// TwinCAT 3 PLC project OOP_Curso
// ProgramVersion: 3.1.4023.0
// libraries:
//   Tc2_Standard, * (Beckhoff Automation GmbH)
//   Tc2_System, * (Beckhoff Automation GmbH)
//   Tc2_Utilities, * (Beckhoff Automation GmbH)
//   Tc3_Module, * (Beckhoff Automation GmbH)
// project tree:
//   02_Clases_Y_Objetos/Clase/ Coche.TcPOU
//   02_Clases_Y_Objetos/ _02_Clase_y_Objetos.TcPOU
//   03_Clases_Y_Objetos/Clase/ Coche_3.TcPOU
//   03_Clases_Y_Objetos/ _03_Clase_y_Objetos.TcPOU
//   04_Clases_Y_Objetos/Clase/ fb_tipos_de_datos.TcPOU
//   04_Clases_Y_Objetos/ GVL4.TcGVL, _04_Clases_y_Objetos.TcPOU
//   05_Metodo/ fbreturn5.TcPOU, FB_ejemplo_Method.TcPOU, interface3.TcIO, ST_sample2.TcDUT, _05_Metodo.TcPOU
//   06_Propiedad/ FB_ejemplo_Propiedad.TcPOU, ST_Property.TcDUT, _06_Propiedad.TcPOU
//   07_Herencia_FB/ FB_Hijo.TcPOU (not stored), FB_Padre.TcPOU, Motor.TcPOU (not stored), Pump.TcPOU (not stored), _07_Herencia.TcPOU (not stored)
//   08_Herencia_Estructura_y_Interface/Herencia_Estructura/ ST_1.TcDUT, ST_2.TcDUT, ST_Base1.TcDUT, ST_Sub1.TcDUT, ST_Sub2.TcDUT
//   08_Herencia_Estructura_y_Interface/Herencia_Interface/ FB_Sub1.TcPOU, FB_Sub2.TcPOU, I_Base1.TcIO, I_Base2.TcIO, I_Sub1.TcIO, I_Sub2.TcIO
//   08_Herencia_Estructura_y_Interface/ _08_Herencia_Estructura_y_Interface.TcPOU
//   09_THIS_SUPER/SUPER/ FB_1.TcPOU, FB_Base.TcPOU
//   09_THIS_SUPER/THIS/ FB_A.TcPOU, FB_B.TcPOU, F_FunA.TcPOU
//   09_THIS_SUPER/ _09_THIS_SUPER.TcPOU
//   10_Interface/Interface1/ FB_Sensor.TcPOU, I_Sensor.TcIO
//   10_Interface/Interface2/ FB_TestA.TcPOU, FB_TestB.TcPOU, ITF_MyTest.TcIO, myFC.TcPOU
//   10_Interface/ _10_Interface.TcPOU
//   11_Puntero_y_Referencia/ Fc_AreaCalcPoint.TcPOU, Fc_AreaCalcRef.TcPOU, Fc_AreaCalcVal.TcPOU, Fc_AverageReferencia.TcPOU, Fc_AverageValues.TcPOU, SR_Main_01.TcPOU, SR_Main_02.TcPOU, SR_Main_03.TcPOU, SR_Main_04.TcPOU, stMotorCtrl.TcDUT, st_Rectangulo.TcDUT, _11_Puntero_y_Referencia.TcPOU
//   13_FB_Abstracto_vs_Interface/1_FB_Abstracto/ ClassDiagram.TcCD (not stored), FB_ContractEmployee.TcPOU (not stored), FB_Employee.TcPOU (not stored), FB_FullTimeEmployee.TcPOU, _13_1_Main_Abstract.TcPOU
//   13_FB_Abstracto_vs_Interface/2_Interfaz/ ClassDiagram_1.TcCD (not stored), FB_ContractEmployee_1.TcPOU (not stored), FB_FullTimeEmployee_1.TcPOU (not stored), I_Employee.TcIO (not stored), _13_2_Main_Interfaz.TcPOU
//   13_FB_Abstracto_vs_Interface/3_Combinacion/ ClassDiagram_2.TcCD (not stored), FB_ContractEmployee_2.TcPOU, FB_Employee_1.TcPOU (not stored), FB_FullTimeEmployee_2.TcPOU (not stored), I_Employee_1.TcIO (not stored), _13_3_Main_Combinacion.TcPOU
//   12_Concepto Keyword Abstract/ AbstractLoadCell.TcPOU, AbstractLogger.TcPOU, ConcreteADSLogger.TcPOU, ConcreteCSVLogger.TcPOU, ConcreteLoadCell.TcPOU, _12_Concepto_Keyword_Abstract.TcPOU
//   14_Interface_Fluida/14_1/ FB_Calculate.TcPOU, I_Calculate.TcIO
//   14_Interface_Fluida/14_2/ FB_Calcul.TcPOU, I_Clear.TcIO, I_Operation.TcIO, I_SetNumber.TcIO
//   14_Interface_Fluida/ _14_Interface_Fluida.TcPOU
//   15_Interface_vs_Herencia/ ClassDiagram_3.TcCD (not stored), FB_NivelSensor.TcPOU, FB_Pump.TcPOU, I_Analog.TcIO, I_Run.TcIO, FB_UltraSonicSensor.TcPOU, FB_VFD.TcPOU, _15_Interface_vs_Herencia.TcPOU
//   16_17_Interface_vs_Herencia/ FB_MyLight1.TcPOU, _16_Interface_vs_Herencia.TcPOU (not stored)
//   16_17_Interface_vs_Herencia/PLC-Library/Clases/ FB_DelayedLight.TcPOU (not stored), FB_DimmingLight.TcPOU (not stored), FB_Light.TcPOU, FB_RoomController.TcPOU (not stored)
//   16_17_Interface_vs_Herencia/PLC-Library/ ClassDiagram_4.TcCD (not stored), FB_MyLight.TcPOU
//   16_17_Interface_vs_Herencia/PLC-Library/Interfaces/ I_Delayable.TcIO, I_Dimmable.TcIO (not stored), I_Light.TcIO (not stored)
//   16_17_Interface_vs_Herencia/Tests/ P_DelayedLight_Test_CFC.TcPOU (not stored), P_DelayedLight_Test_ST.TcPOU (not stored), P_DimmingLight_Test_CFC.TcPOU, P_DimmingLight_Test_ST.TcPOU (not stored), P_Light_Test_CFC.TcPOU, P_Light_Test_ST.TcPOU, P_MyLight_Test_CFC.TcPOU, P_MyLight_Test_ST.TcPOU, P_RoomController_Test_CFC.TcPOU, P_RoomController_Test_ST.TcPOU
//   17_Otros_Operadores_1/ ST_Estructura.TcDUT (not stored), _17_Otros_Operadores1.TcPOU
//   18_Otros_Operadores_2/TestAndSet/ GVL.TcGVL, TestAndSet1.TcPOU
//   18_Otros_Operadores_2/ _18_Otros_Operadores2.TcPOU
//   18_Otros_Operadores_2/__QUERYPOINTER/ FB_Variante.TcPOU, I_Base.TcIO, I_Derived.TcIO, QUERYPOINTER.TcPOU
//   18_Otros_Operadores_2/__TRY__CATCH/ GVL_Exc.TcGVL, F_SaveExceptionCode.TcPOU, TRY_CATCH.TcPOU
//   18_Otros_Operadores_2/__VARINFO/ VARINFO.TcPOU
//   19_ExST/ _19_ExST.TcPOU
//   24_SOLID_SRP/Clases_SRP/ FB_Empleado.TcPOU (not stored), FB_RegistroDeTiempo.TcPOU
//   24_SOLID_SRP/ Class Diagram_SOLID_SRP.TcCD (not stored), _24_SOLID_SRP.TcPOU
//   24_SOLID_SRP/Estructuras_SRP/ ST_Empleado.TcDUT (not stored), ST_Horario.TcDUT, ST_RegistroDeTiempoEmpleado.TcDUT
//   25_SOLID_OCP/Clases_OCP/ FB_Coche.TcPOU, FB_Moto.TcPOU, FB_Vehiculo.TcPOU
//   25_SOLID_OCP/ Class Diagram_SOLID_OCP.TcCD (not stored), _25_SOLID_OCP.TcPOU
//   26_SOLID_LSP/Clases_LSP/ Coche1.TcPOU, Conductor.TcPOU, Moto1.TcPOU, Vehiculo.TcPOU
//   26_SOLID_LSP/ Class Diagram_SOLID_LSP.TcCD (not stored), _26_SOLID_LSP.TcPOU
//   26_SOLID_LSP/Interfaces_LSP/ I_Mover.TcIO
//   27_SOLID_ISP/Clases_ISP/ Aguila.TcPOU, Avestruz.TcPOU, Pato.TcPOU
//   27_SOLID_ISP/ Class Diagram_SOLID_ISP.TcCD (not stored), _27_SOLID_ISP.TcPOU
//   27_SOLID_ISP/Interfaces_ISP/ I_AveCorredora.TcIO, I_AveNadadora.TcIO, I_AveVoladora.TcIO
//   28_SOLID_DIP/Clases_DIP/ ConexionEthernet.TcPOU, ConexionSerial.TcPOU, Dispositivo.TcPOU
//   28_SOLID_DIP/ ClassDiagram_SOLID_DIP.TcCD (not stored), _28_SOLID_DIP.TcPOU
//   28_SOLID_DIP/Interfaces_DIP/ I_Conexion.TcIO
//   30_UML_ClassDiagram/ 30_UML_ClassDiagram.TcCD (not stored), GVL_1.TcGVL, ITF_Profesor.TcIO, Persona.TcPOU, Profesor.TcPOU
//   31_UML_relaciones/ ClassDiagram_UML_Relaciones.TcCD (not stored), Corazon.TcPOU, Hombre.TcPOU, Humano.TcPOU, I_Humano.TcIO, Sangre.TcPOU
//   32_UML_StateChart/32_VISU/ _32_Visualization.TcVIS
//   32_UML_StateChart/ Kaffemaschine.TcPOU
//   32_UML_StateChart/32_POUs/ FB_UML_SC.TcPOU, _32_MAIN.TcPOU
//   / Gestor de visualización.TcVMO (not stored), GlobalTextList.TcGTLO, PlcTask.TcTTO
//   _MAIN/ MAIN.TcPOU
// real-time tasks:
//   TASK PlcTask: cycle T#10ms, priority 20, ADS port 350

CONFIGURATION OOP_Curso
    RESOURCE PLC ON TwinCAT3
        TASK PlcTask(INTERVAL := T#10ms, PRIORITY := 20);
        PROGRAM MAIN WITH PlcTask : MAIN;
    END_RESOURCE
END_CONFIGURATION

// ---- 05_Metodo/ST_sample2.TcDUT
TYPE ST_sample2 :
STRUCT
	bbool	: BOOL;
	bVar 	: BOOL;
    nVar 	: INT;
	rreal 	: REAL;
	sstring : STRING;
END_STRUCT
END_TYPE

// ---- 06_Propiedad/ST_Property.TcDUT
TYPE ST_Property :
STRUCT
	b1,b2,b3 : BOOL;
	r1,r2,r3 : REAL;	
END_STRUCT
END_TYPE

// ---- 08_Herencia_Estructura_y_Interface/Herencia_Estructura/ST_1.TcDUT
TYPE ST_1:
STRUCT
	sStruct : ST_2;
	sstring : STRING(80);
END_STRUCT
END_TYPE

// ---- 08_Herencia_Estructura_y_Interface/Herencia_Estructura/ST_2.TcDUT
TYPE ST_2 :
STRUCT
	bBool : BOOL;
END_STRUCT
END_TYPE

// ---- 08_Herencia_Estructura_y_Interface/Herencia_Estructura/ST_Base1.TcDUT
TYPE ST_Base1 :
STRUCT
	bBool1: BOOL;
	iINT : INT;
	rReal : REAL;	
END_STRUCT
END_TYPE

// ---- 08_Herencia_Estructura_y_Interface/Herencia_Estructura/ST_Sub1.TcDUT
TYPE ST_Sub1 EXTENDS ST_Base1:
STRUCT
	ttime :TIME;
	tton  : TON;
END_STRUCT
END_TYPE

// ---- 08_Herencia_Estructura_y_Interface/Herencia_Estructura/ST_Sub2.TcDUT
TYPE ST_Sub2 EXTENDS ST_Sub1 :
STRUCT
	bBool2: BOOL;
END_STRUCT
END_TYPE

// ---- 11_Puntero_y_Referencia/stMotorCtrl.TcDUT
TYPE stMotorCtrl :
STRUCT
	rTpoAcelDecel :REAL; // Tiempo para acelerar/decelerar hasta alcanazar la velocidad.
	rVelRpm       :REAL; // Velocidad en RPM.
	xMotorOff     :BOOL; // Bit de paro ON.
	xMotorOn      :BOOL   ; // Bit de marcha OFF.	
END_STRUCT
END_TYPE

// ---- 11_Puntero_y_Referencia/st_Rectangulo.TcDUT
TYPE st_Rectangulo :
STRUCT
   rASide    	: REAL; // Parámetro de entrada que contiene el lado A del rectangulo.
   rBSide    	: REAL; // Parámetro de entrada que contiene el lado B del rectangulo.	
   rArea		: REAL; // Valor del area
END_STRUCT
END_TYPE

// ---- 24_SOLID_SRP/Estructuras_SRP/ST_Horario.TcDUT
TYPE ST_Horario :
STRUCT
	HoraEntrada : DATE_AND_TIME;
    HoraSalida : DATE_AND_TIME;
END_STRUCT
END_TYPE

// ---- 24_SOLID_SRP/Estructuras_SRP/ST_RegistroDeTiempoEmpleado.TcDUT
TYPE ST_RegistroDeTiempoEmpleado :
STRUCT
	stEmpleado : ST_Empleado; // Datos de la función Empleado
    stHorario  : ST_Horario;
END_STRUCT
END_TYPE

// ---- 04_Clases_Y_Objetos/GVL4.TcGVL
//{attribute 'qualified_only'}
VAR_GLOBAL
	 nVarExt1 : INT; // 1st external variable
END_VAR

// ---- 18_Otros_Operadores_2/TestAndSet/GVL.TcGVL
{attribute 'qualified_only'}
VAR_GLOBAL
    bGlobalTestFlag : BOOL;
END_VAR

// ---- 18_Otros_Operadores_2/__TRY__CATCH/GVL_Exc.TcGVL
{attribute 'qualified_only'}
VAR_GLOBAL CONSTANT
    cMaxExc            : UINT := 10;
END_VAR
VAR_GLOBAL
    nExcIndex          : UINT;
    aExceptionHistory  : ARRAY[0..cMaxExc] OF __SYSTEM.ExceptionCode;
END_VAR

// ---- 30_UML_ClassDiagram/GVL_1.TcGVL
{attribute 'qualified_only'}
VAR_GLOBAL
	variable1 : BOOL;
	VarInt: INT;
END_VAR

// ---- 05_Metodo/interface3.TcIO
INTERFACE interface3

METHOD itf_metodo : BOOL
VAR_INPUT
END_VAR
END_METHOD

PROPERTY itf_propiedad : real
GET
END_GET
SET
END_SET
END_PROPERTY

END_INTERFACE

// ---- 08_Herencia_Estructura_y_Interface/Herencia_Interface/I_Base1.TcIO
INTERFACE I_Base1

METHOD metodo_base1 : BOOL
VAR_INPUT
END_VAR
END_METHOD

PROPERTY Prop_base1 : bool
GET
END_GET
SET
END_SET
END_PROPERTY

END_INTERFACE

// ---- 08_Herencia_Estructura_y_Interface/Herencia_Interface/I_Base2.TcIO
INTERFACE I_Base2

METHOD metodo_base2 : BOOL
VAR_INPUT
END_VAR
END_METHOD

PROPERTY Prop_base2 : bool
GET
END_GET
SET
END_SET
END_PROPERTY

END_INTERFACE

// ---- 08_Herencia_Estructura_y_Interface/Herencia_Interface/I_Sub1.TcIO
INTERFACE I_Sub1 EXTENDS I_Base1, I_Base2

METHOD metodo_sub1 : BOOL
VAR_INPUT
END_VAR
END_METHOD

PROPERTY Prop_sub1 : BOOL
GET
END_GET
SET
END_SET
END_PROPERTY

END_INTERFACE

// ---- 08_Herencia_Estructura_y_Interface/Herencia_Interface/I_Sub2.TcIO
INTERFACE I_Sub2 EXTENDS I_Sub1

METHOD metodo_sub2 : BOOL
VAR_INPUT
END_VAR
END_METHOD

PROPERTY Prop_sub2 : BOOL
GET
END_GET
SET
END_SET
END_PROPERTY

END_INTERFACE

// ---- 10_Interface/Interface1/I_Sensor.TcIO
INTERFACE I_Sensor

PROPERTY Calibrado : BOOL
GET
END_GET
END_PROPERTY

METHOD Calibrar
END_METHOD

PROPERTY Consigna : REAL
SET
END_SET
END_PROPERTY


METHOD Descalibrar
END_METHOD

METHOD LeerValor : INT
END_METHOD

PROPERTY Temperatura : REAL
GET
END_GET
END_PROPERTY

END_INTERFACE

// ---- 10_Interface/Interface2/ITF_MyTest.TcIO
INTERFACE ITF_MyTest

METHOD METH1 : BOOL
VAR_INPUT
END_VAR
END_METHOD

METHOD METH2 : STRING
VAR_INPUT
END_VAR
END_METHOD

METHOD METH3 : REAL
VAR_INPUT
END_VAR
END_METHOD

PROPERTY Prop1 : BOOL
GET
END_GET
SET
END_SET
END_PROPERTY

PROPERTY Prop2 : REAL
GET
END_GET
SET
END_SET
END_PROPERTY

PROPERTY Prop3 : STRING
GET
END_GET
SET
END_SET
END_PROPERTY

END_INTERFACE

// ---- 14_Interface_Fluida/14_1/I_Calculate.TcIO
INTERFACE I_Calculate

METHOD Clear : I_Calculate
END_METHOD

METHOD DecreaseBy : I_Calculate
VAR_INPUT
	lDecreaseBy : REAL;
END_VAR
END_METHOD

METHOD DivideBy : I_Calculate
VAR_INPUT
	lDivideBy : REAL;
END_VAR
END_METHOD

METHOD GetResult : LREAL
VAR_INPUT
END_VAR
END_METHOD

METHOD IncreaseBy : I_Calculate
VAR_INPUT
	lIncreaseBy : REAL;
END_VAR
END_METHOD

METHOD MultiplyBy : I_Calculate
VAR_INPUT
	lMultiplyBy : REAL;
END_VAR
END_METHOD

METHOD SetNumber : I_Calculate
VAR_INPUT
	lNumber : LREAL;
END_VAR
END_METHOD

END_INTERFACE

// ---- 14_Interface_Fluida/14_2/I_Clear.TcIO
INTERFACE I_Clear

METHOD Clear : I_SetNumber
END_METHOD

END_INTERFACE

// ---- 14_Interface_Fluida/14_2/I_Operation.TcIO
INTERFACE I_Operation EXTENDS I_SetNumber


METHOD DecreaseBy : I_Operation
VAR_INPUT
	lDecreaseBy : REAL;
END_VAR
END_METHOD


METHOD DivideBy : I_Operation
VAR_INPUT
	lDivideBy : REAL;
END_VAR
END_METHOD


METHOD GetResult : LREAL
END_METHOD

METHOD IncreaseBy : I_Operation
VAR_INPUT
	lIncreaseBy : REAL;
END_VAR
END_METHOD


METHOD MultiplyBy : I_Operation
VAR_INPUT
	lMultiplyBy : REAL;
END_VAR
END_METHOD

END_INTERFACE

// ---- 14_Interface_Fluida/14_2/I_SetNumber.TcIO
INTERFACE I_SetNumber

METHOD SetNumber : I_Operation
VAR_INPUT
	lNumber : LREAL;
END_VAR
END_METHOD

END_INTERFACE

// ---- 15_Interface_vs_Herencia/I_Analog.TcIO
INTERFACE I_Analog

PROPERTY AnalogSignal : INT
GET
END_GET
SET
END_SET
END_PROPERTY

METHOD Scale : BOOL
VAR_INPUT
END_VAR
END_METHOD

PROPERTY ScaledAnalog : INT
GET
END_GET
SET
END_SET
END_PROPERTY

END_INTERFACE

// ---- 15_Interface_vs_Herencia/I_Run.TcIO
INTERFACE I_Run

PROPERTY Coil : BOOL
GET
END_GET
SET
END_SET
END_PROPERTY

METHOD Start : BOOL
VAR_INPUT
END_VAR
END_METHOD

METHOD Stop : BOOL
VAR_INPUT
END_VAR
END_METHOD

END_INTERFACE

// ---- 16_17_Interface_vs_Herencia/PLC-Library/Interfaces/I_Delayable.TcIO
INTERFACE I_Delayable EXTENDS __SYSTEM.IQueryInterface

PROPERTY tOffDelay : TIME
GET
END_GET
SET
END_SET
END_PROPERTY

PROPERTY tOnDelay : TIME
GET
END_GET
SET
END_SET
END_PROPERTY

END_INTERFACE

// ---- 18_Otros_Operadores_2/__QUERYPOINTER/I_Base.TcIO
INTERFACE I_Base EXTENDS __SYSTEM.IQueryInterface

METHOD Base : BOOL
VAR_INPUT
END_VAR
END_METHOD

END_INTERFACE

// ---- 18_Otros_Operadores_2/__QUERYPOINTER/I_Derived.TcIO
INTERFACE I_Derived EXTENDS I_Base

METHOD Derived : BOOL
VAR_INPUT
END_VAR
END_METHOD

END_INTERFACE

// ---- 26_SOLID_LSP/Interfaces_LSP/I_Mover.TcIO
INTERFACE I_Mover

METHOD Mover : REAL
VAR_INPUT
	Velocidad_Deseada : REAL;
END_VAR
END_METHOD

END_INTERFACE

// ---- 27_SOLID_ISP/Interfaces_ISP/I_AveCorredora.TcIO
INTERFACE I_AveCorredora

METHOD Correr : BOOL
END_METHOD

END_INTERFACE

// ---- 27_SOLID_ISP/Interfaces_ISP/I_AveNadadora.TcIO
INTERFACE I_AveNadadora

METHOD Nadar : BOOL
END_METHOD

END_INTERFACE

// ---- 27_SOLID_ISP/Interfaces_ISP/I_AveVoladora.TcIO
INTERFACE I_AveVoladora

METHOD Volar : BOOL
END_METHOD

END_INTERFACE

// ---- 28_SOLID_DIP/Interfaces_DIP/I_Conexion.TcIO
INTERFACE I_Conexion

METHOD EstablecerConexion : BOOL
VAR_INPUT
END_VAR
END_METHOD

END_INTERFACE

// ---- 30_UML_ClassDiagram/ITF_Profesor.TcIO
INTERFACE ITF_Profesor

METHOD Fichar
VAR_INPUT
END_VAR
END_METHOD

PROPERTY Salida : int
GET
END_GET
SET
END_SET
END_PROPERTY

END_INTERFACE

// ---- 31_UML_relaciones/I_Humano.TcIO
INTERFACE I_Humano

METHOD Correr
VAR_INPUT
END_VAR
END_METHOD

PROPERTY Nombre : STRING
GET
END_GET
SET
END_SET
END_PROPERTY

END_INTERFACE

// ---- _MAIN/MAIN.TcPOU
PROGRAM MAIN
VAR
END_VAR

// Video de Youtube 02:
_02_Clase_y_Objetos();

// Video de Youtube 03:
_03_Clase_y_Objetos();

// Video de Youtube 04:
_04_Clases_y_Objetos();

// Video de Youtube 05;
_05_Metodo();

// Video de Youtube 06;
_06_Propiedad();

// Video de Youtube 07;
_07_Herencia();

// Video de Youtube 08;
_08_Herencia_Estructura_y_Interface();

// Video de Youtube 09;
_09_THIS_SUPER();

// Video de Youtube 10;
_10_Interface();

// Video de Youtube 11;
_11_Puntero_y_Referencia();

// Video de Youtube 12;
_12_Concepto_Keyword_Abstract();

// Video de Youtube 13;
_13_1_Main_Abstract();
_13_2_Main_Interfaz();
_13_3_Main_Combinacion();

// Video de Youtube 14;
_14_Interface_Fluida();

// Video de Youtube 15:
_15_Interface_vs_Herencia();

// Video de Youtube 16:
_16_Interface_vs_Herencia();

// Video de Youtube 17:
_17_Otros_Operadores1();

// Video de Youtube 18:
_18_Otros_Operadores2();

// Video de Youtube 19:
_19_ExST();

// Video de Youtube 24
_24_SOLID_SRP();

// Video de Youtube 25
_25_SOLID_OCP();

// Video de Youtube 26
_26_SOLID_LSP();

// Video de Youtube 27
_27_SOLID_ISP();

// Video de Youtube 28
_28_SOLID_DIP();

// Video de Youtube 32
_32_MAIN();

END_PROGRAM

// ---- 02_Clases_Y_Objetos/_02_Clase_y_Objetos.TcPOU
PROGRAM _02_Clase_y_Objetos
VAR
	// tenemos la Clase Coche y la instanciamos y obtenemos los Objetos: Mercedes, Bmw y Audi.
	Mercedes : Coche;
	Bmw : Coche;
	Audi: Coche;
	
	Color : STRING;
	Marca : STRING;
	
	Acelerar : BOOL;
	Conducir:  BOOL;
	Frenar  : BOOL;
	
	
END_VAR

//Objeto Mercedes
//llamadas a sus métodos.
IF Acelerar THEN
	Mercedes.Acelerar();
	Acelerar := FALSE;
END_IF

IF Conducir THEN
	Mercedes.Conducir();
	Conducir := FALSE;
END_IF

IF Frenar THEN
	Mercedes.Frenar();
	Frenar := FALSE;
END_IF

//llamadas a sus propiedades.
Mercedes.Marca := 'Mercedes';
Mercedes.Color := 'Negro';
Color := Mercedes.Color;

END_PROGRAM

// ---- 02_Clases_Y_Objetos/Clase/Coche.TcPOU
FUNCTION_BLOCK Coche
VAR_INPUT 
END_VAR
VAR_OUTPUT
END_VAR
VAR
	_Marca : STRING;
	_Color : STRING;
	accion : STRING;
END_VAR

METHOD PUBLIC Acelerar
accion := 'acelerar';
END_METHOD

PROPERTY PUBLIC Color : STRING
GET
Color := _Color;
END_GET
SET
_Color := Color;
END_SET
END_PROPERTY

METHOD PUBLIC Conducir
accion := 'conducir';
END_METHOD

METHOD PUBLIC Frenar
accion := 'frenar';
END_METHOD

PROPERTY PUBLIC Marca : STRING
GET
Marca := _Marca;
END_GET
SET
_Marca := Marca;
END_SET
END_PROPERTY

END_FUNCTION_BLOCK

// ---- 03_Clases_Y_Objetos/_03_Clase_y_Objetos.TcPOU
PROGRAM _03_Clase_y_Objetos
VAR
	// tenemos la Clase Coche y la instanciamos y obtenemos los Objetos: Mercedes, Bmw y Audi.
	Mercedes : Coche_3(Marca:= 'Mercedes', Color := 'Azul');
	
	Color : STRING;
	Marca : STRING;
	
	Acelerar : BOOL;
	Conducir:  BOOL;
	Frenar  : BOOL;
	
	CambiarColor : BOOL;
END_VAR

//Objeto Mercedes
//llamadas a sus métodos.
IF Acelerar THEN
	Mercedes.Acelerar();
	Acelerar := FALSE;
END_IF

IF Conducir THEN
	Mercedes.Conducir();
	Conducir := FALSE;
END_IF

IF Frenar THEN
	Mercedes.Frenar();
	Frenar := FALSE;
END_IF

//llamadas a sus propiedades.
//Mercedes.Marca := 'Mercedes';
IF CambiarColor THEN
	Mercedes.Color := 'Negro';
	CambiarColor := FALSE;
END_IF

Color := Mercedes.Color;

END_PROGRAM

// ---- 03_Clases_Y_Objetos/Clase/Coche_3.TcPOU
FUNCTION_BLOCK Coche_3
VAR_INPUT
	bInput : BOOL;
END_VAR
VAR_OUTPUT
	bOutput : BOOL;
END_VAR
VAR_IN_OUT
	bInOut : BOOL;
END_VAR
VAR
	_Marca : STRING;
	_Color : STRING;
	accion : STRING;
END_VAR

METHOD PUBLIC Acelerar
accion := 'acelerar';
END_METHOD

PROPERTY PUBLIC Color : STRING
GET
Color := _Color;
END_GET
SET
_Color := Color;
END_SET
END_PROPERTY

METHOD PUBLIC Conducir
accion := 'conducir';
END_METHOD

METHOD FB_exit : BOOL
VAR_INPUT
	bInCopyCode : BOOL; // if TRUE, the exit method is called for exiting an instance that is copied afterwards (online change).
END_VAR
END_METHOD

METHOD FB_init : BOOL
VAR_INPUT
	bInitRetains : BOOL; // if TRUE, the retain variables are initialized (warm start / cold start)
	bInCopyCode : BOOL;  // if TRUE, the instance afterwards gets moved into the copy code (online change)
	Marca        : STRING;
	Color        : STRING;
END_VAR
THIS^._Marca := Marca;
THIS^._Color := Color;
END_METHOD

METHOD FB_reinit : BOOL
VAR_INPUT
END_VAR
END_METHOD

METHOD PUBLIC Frenar
accion := 'frenar';
END_METHOD

PROPERTY PUBLIC Marca : STRING
GET
Marca := _Marca;
END_GET
SET
_Marca := Marca;
END_SET
END_PROPERTY

END_FUNCTION_BLOCK

// ---- 04_Clases_Y_Objetos/_04_Clases_y_Objetos.TcPOU
PROGRAM _04_Clases_y_Objetos
VAR
	fb :fb_tipos_de_datos;
	binput : BOOL;
	in_out1 : LINT;
	in_out_constant1 : DINT := 10;
END_VAR


fb(
//	binput:= binput, 
//	binput2:= , 
//	output1=> , 
	in_out1:= in_out1, 
	in_out_constant1:= in_out_constant1 );

END_PROGRAM

// ---- 04_Clases_Y_Objetos/Clase/fb_tipos_de_datos.TcPOU
FUNCTION_BLOCK fb_tipos_de_datos
VAR_INPUT
	binput : BOOL;
END_VAR
VAR_INPUT
	binput2 : BOOL;
END_VAR
VAR_OUTPUT
	output1 : REAL;
END_VAR
VAR_IN_OUT
	in_out1 : LINT;
END_VAR
VAR_IN_OUT CONSTANT
	in_out_constant1 : DINT;
END_VAR
VAR
	var1 : STRING;
END_VAR
VAR_TEMP
	temp1 : ULINT;
END_VAR
VAR_STAT
    nVarStat1 : INT;
	aarray  : ARRAY[1..n] OF INT;
END_VAR
VAR_EXTERNAL
    nVarExt1 : INT; // 1st external variable
END_VAR
VAR PERSISTENT
    nVarPers1 : DINT; (* 1. Persistent variable *)
    bVarPers2 : BOOL; (* 2. Persistent variable *)
END_VAR
VAR RETAIN
    nRem1 : INT;
END_VAR
VAR CONSTANT
	n : INT:= 10;
END_VAR

END_FUNCTION_BLOCK

// ---- 05_Metodo/_05_Metodo.TcPOU
PROGRAM _05_Metodo
VAR
	fbejemplo_metodo : FB_ejemplo_Method;
	
	bPonerAUnobBoolfb : BOOL;
	bPonerACerobBoolfb: BOOL;
	
	bBool : BOOL;
	statusbBool : BOOL;
	bPonerAUnobBool : BOOL;
	bPonerACerobBool: BOOL;
	
	nSingleGet  : INT;
    stGet       : ST_Sample2;    
    bSet        : BOOL;
    stSet       : ST_Sample2;
	
	counter : INT;
	outvarcounter: INT;
END_VAR

IF 	bPonerAUnobBoolfb THEN
	bPonerAUnobBoolfb := FALSE;
	fbejemplo_metodo.metodo1_a_Uno_bBool();	
END_IF


IF 	bPonerACerobBoolfb THEN
	bPonerACerobBoolfb := FALSE;
	fbejemplo_metodo.metodo1_a_cero_bBool();
END_IF


IF 	bPonerAUnobBool THEN
	bPonerAUnobBool := FALSE;
	statusbBool := fbejemplo_metodo.metodo1_a_Uno_InOut(bBool);
END_IF

IF 	bPonerACerobBool THEN
	bPonerACerobBool := FALSE;
	statusbBool := fbejemplo_metodo.metodo1_a_Cero_InOut(bBool);
END_IF

// ejemplo para declarar variables lo mas cerca posible del metodo: declaración dentro del metodo de variable con VAR_INST :
counter := fbejemplo_metodo.Metodo4_VarInst(outvarcounter=>outvarcounter);

// Set and Get
IF bSet THEN  
	nSingleGet := fbejemplo_metodo.metodo2_struct(stSet).nVar;
	stGet      := fbejemplo_metodo.metodo2_struct(stSet);
	bSet            := FALSE;
END_IF

END_PROGRAM

// ---- 05_Metodo/FB_ejemplo_Method.TcPOU
FUNCTION_BLOCK FB_ejemplo_Method
VAR_INPUT
END_VAR
VAR_OUTPUT
END_VAR
VAR
	bBool : BOOL;
	ststruct : ST_sample2;
	fb5 : fbreturn5;
END_VAR

METHOD metodo0_Declaracion_variables
VAR_INPUT
	binput : BOOL;
END_VAR
VAR_INPUT
	binput2 : BOOL;
END_VAR
VAR_OUTPUT
	output1 : REAL;
END_VAR
VAR_IN_OUT
	in_out1 : LINT;
END_VAR
VAR_IN_OUT CONSTANT
	in_out_constant1 : DINT;
END_VAR
VAR
	var1 : STRING;
END_VAR
//!!! no se pueden declarar variables TEMPORALES dentro de la zona de declaración de variables del método!!!
//VAR_TEMP
//	temp1 : ULINT;
//END_VAR
VAR_INST
	counter : INT;
END_VAR
VAR_STAT
    nVarStat1 : INT;
	aarray  : ARRAY[1..n] OF INT;
END_VAR
VAR_EXTERNAL
    nVarExt1 : INT; // 1st external variable
END_VAR
//!!! no se pueden declarar variables PERSISTENT ni RETAIN dentro de la zona de declaración de variables del método!!!
//VAR PERSISTENT
//    nVarPers1 : DINT; (* 1. Persistent variable *)
//    bVarPers2 : BOOL; (* 2. Persistent variable *)
//END_VAR
//VAR RETAIN
//    nRem1 : INT;
//END_VAR
VAR CONSTANT
	n : INT:= 10;
END_VAR
END_METHOD

METHOD metodo1_a_Cero_bBool
THIS^.bBool := false;
END_METHOD

METHOD metodo1_a_Cero_InOut : bool
VAR_IN_OUT
	bBool : BOOL;
END_VAR
// Método que pone a 0 la variable definida en in_Out
bBool := FALSE;
// return value bBOOL
metodo1_a_Cero_InOut := FALSE;
END_METHOD

METHOD metodo1_a_Uno_bBool
THIS^.bBool := true;
END_METHOD

METHOD metodo1_a_Uno_InOut : BOOL
VAR_IN_OUT
	bBool : BOOL;
END_VAR
// Método que pone a 1 la variable definida en in_Out
bBool := TRUE;
// return value bBOOL
metodo1_a_Uno_InOut := TRUE;
END_METHOD

METHOD PUBLIC metodo2_struct : REFERENCE TO ST_sample2
VAR_INPUT
	st_struct : ST_sample2;
END_VAR


THIS^.ststruct := st_struct;

metodo2_struct REF= THIS^.ststruct;
END_METHOD

METHOD PRIVATE metodo3_interface : interface3
VAR_INPUT
END_VAR
END_METHOD

METHOD Metodo4_VarInst : INT
VAR_OUTPUT
	outvarcounter : INT;
END_VAR
VAR
	varcounter : INT;
END_VAR
VAR_INST
	counter : INT;
END_VAR
counter := counter + 1;
Metodo4_VarInst := counter;

varcounter := varcounter + 1; 
outvarcounter := varcounter;
END_METHOD

METHOD metodo5_returnfb : fbreturn5
VAR_INPUT
END_VAR
metodo5_returnfb := fb5;
END_METHOD

END_FUNCTION_BLOCK

// ---- 05_Metodo/fbreturn5.TcPOU
FUNCTION_BLOCK fbreturn5
VAR_INPUT
END_VAR
VAR_OUTPUT
END_VAR
VAR
END_VAR

END_FUNCTION_BLOCK

// ---- 06_Propiedad/_06_Propiedad.TcPOU
PROGRAM _06_Propiedad
VAR
	myFBProperty : FB_Ejemplo_Propiedad;
	
	bSet1, bSet2 : BOOL;
	
	IntData 	: INT;
	BoolData 	: BOOL;
	GetSTData 	: ST_Property;
	SetSTData 	: ST_Property;
	ioData    	: INT;
	counter   	: INT;
	
	myValueMultiply : INT;
END_VAR

IF bSet1 THEN
	bSet1:= FALSE;
	myFBProperty.ValueBool := TRUE;
	myFBProperty.ValueInt := 123;
	SetSTData.b1 := TRUE;
	SetSTData.b2 := FALSE;
	SetSTData.b3 := FALSE;
	SetSTData.r1 := 1.0;
	SetSTData.r2 := 2.0;
	SetSTData.r3 := 3.0;

END_IF

IF bSet2 THEN
	bSet2:= FALSE;
	myFBProperty.ValueBool := FALSE;
	myFBProperty.ValueInt := 456;
	SetSTData.b1 := FALSE;
	SetSTData.b2 := TRUE;
	SetSTData.b3 := TRUE;
	SetSTData.r1 := 11.0;
	SetSTData.r2 := 22.0;
	SetSTData.r3 := 33.0;
END_IF

IntData := 	myFBProperty.ValueInt;
BoolData := myFBProperty.ValueBool;

//STRUCT
GetSTData.b1 := myFBProperty.ValueST.b1;
GetSTData.r1 := myFBProperty.ValueST.r1;

myFBProperty.ValueST := SetSTData;

//IN_OUT;
IF counter < 0 OR counter > 9999 THEN
	counter := 1;
ELSE
	counter := counter + 1;
END_IF

//myFBProperty(myIN_OUT:=counter);
//myFBProperty.Value_INT_OUT := 120;
ioData := myFBProperty.Value_INT_OUT;
myFBProperty(myIN_OUT:=counter);

myFBProperty.Multiply(2,3);
myValueMultiply := myFBProperty.ValueMultiply;

END_PROGRAM

// ---- 06_Propiedad/FB_ejemplo_Propiedad.TcPOU
FUNCTION_BLOCK FB_ejemplo_Propiedad
VAR_INPUT
END_VAR
VAR_OUTPUT
END_VAR
VAR_IN_OUT
	myIN_OUT : INT;
END_VAR
VAR
	myBool : BOOL;
	myInt : INT;
	myST  : ST_Property;
	myValueMultiply: INT;
END_VAR

METHOD Multiply
VAR_INPUT
	iValueMultiply1 : INT;
	iValueMultiply2 : INT;
END_VAR
myValueMultiply := iValueMultiply1 * iValueMultiply2;
END_METHOD

PROPERTY Value_INT_OUT : INT
GET
IF NOT __ISVALIDREF(myIN_OUT) THEN
	RETURN;
END_IF

Value_INT_OUT := myIN_OUT;
END_GET
SET
myIN_OUT := Value_INT_OUT;
END_SET
END_PROPERTY

PROPERTY ValueBool : BOOL
GET
ValueBool := myBool;
END_GET
SET
 myBool := ValueBool;
END_SET
END_PROPERTY

PROPERTY ValueInt : INT
GET
ValueInt := myint;
END_GET
SET
 myint := ValueInt;
END_SET
END_PROPERTY

PROPERTY ValueMultiply : INT
GET
ValueMultiply := myValueMultiply;
END_GET
END_PROPERTY

PROPERTY ValueST : reference to ST_Property
GET
ValueST REF= myST;
END_GET
SET
IF NOT __ISVALIDREF(ValueST) THEN
	RETURN;
END_IF

myST := ValueST;
END_SET
END_PROPERTY

END_FUNCTION_BLOCK

// ---- 08_Herencia_Estructura_y_Interface/_08_Herencia_Estructura_y_Interface.TcPOU
PROGRAM _08_Herencia_Estructura_y_Interface
VAR
	//Extensión de Estructura:
	stestructura1  : ST_Sub1;
	stestructura2  : ST_Sub2;
	stestructura11 : ST_1;
	
	//Extensión de Interface:
	Sub1 : FB_Sub1;
	Sub2 : FB_Sub2;
	bBool : BOOL;

END_VAR

//Extensión de Estructura:
stestructura1.bBool1;
stestructura1.iINT;
stestructura1.rReal;
stestructura1.ttime;
stestructura1.tton(in:= TRUE, pt:=T#1S);

stestructura2.bBool1;
stestructura2.iINT;
stestructura2.rReal;
stestructura2.ttime;
stestructura2.tton(in:= TRUE, pt:=T#1S);
stestructura2.bBool2;


stestructura11.sstring;
stestructura11.sStruct.bBool;

//Extensión de Interface:
Sub1.metodo_base1();
Sub1.Prop_base1;
Sub1.Prop_base1 := bBool;

Sub2.metodo_sub2();
Sub2.Prop_base2;
Sub1.Prop_base2 := bBool;

END_PROGRAM

// ---- 08_Herencia_Estructura_y_Interface/Herencia_Interface/FB_Sub1.TcPOU
FUNCTION_BLOCK FB_Sub1 IMPLEMENTS I_Sub1
VAR_INPUT
END_VAR
VAR_OUTPUT
END_VAR
VAR
END_VAR

{warning 'Agregar implementación de método'}
METHOD metodo_base1 : BOOL
END_METHOD

{warning 'Agregar implementación de método'}
METHOD metodo_base2 : BOOL
END_METHOD

{warning 'Agregar implementación de método'}
METHOD metodo_sub1 : BOOL
END_METHOD

{warning 'Agregar implementación de propiedad'}
PROPERTY Prop_base1 : BOOL
GET
END_GET
SET
END_SET
END_PROPERTY

{warning 'Agregar implementación de propiedad'}
PROPERTY Prop_base2 : BOOL
GET
END_GET
SET
END_SET
END_PROPERTY

{warning 'Agregar implementación de propiedad'}
PROPERTY Prop_sub1 : BOOL
GET
END_GET
SET
END_SET
END_PROPERTY

END_FUNCTION_BLOCK

// ---- 08_Herencia_Estructura_y_Interface/Herencia_Interface/FB_Sub2.TcPOU
FUNCTION_BLOCK FB_Sub2 IMPLEMENTS I_Sub2
VAR_INPUT
END_VAR
VAR_OUTPUT
END_VAR
VAR
END_VAR

{warning 'Agregar implementación de método'}
METHOD metodo_base1 : BOOL
END_METHOD

{warning 'Agregar implementación de método'}
METHOD metodo_base2 : BOOL
END_METHOD

{warning 'Agregar implementación de método'}
METHOD metodo_sub1 : BOOL
END_METHOD

{warning 'Agregar implementación de método'}
METHOD metodo_sub2 : BOOL
END_METHOD

{warning 'Agregar implementación de propiedad'}
PROPERTY Prop_base1 : BOOL
GET
END_GET
SET
END_SET
END_PROPERTY

{warning 'Agregar implementación de propiedad'}
PROPERTY Prop_base2 : BOOL
GET
END_GET
SET
END_SET
END_PROPERTY

{warning 'Agregar implementación de propiedad'}
PROPERTY Prop_sub1 : BOOL
GET
END_GET
SET
END_SET
END_PROPERTY

{warning 'Agregar implementación de propiedad'}
PROPERTY Prop_sub2 : BOOL
GET
END_GET
SET
END_SET
END_PROPERTY

END_FUNCTION_BLOCK

// ---- 09_THIS_SUPER/_09_THIS_SUPER.TcPOU
PROGRAM _09_THIS_SUPER
VAR
	// Ejemplo para el puntero THIS^
	fbMyfbB : FB_B;
	
	// Ejemplo para el puntero SUPER^
    fbMyBase : FB_Base;
    fbMyFB_1 : FB_1;
    nTHIS    : INT;
    nBase    : INT;	
END_VAR

// Ejemplo para el puntero THIS^
fbMyfbB(nVarA:=0, nVarB:= 0);
fbMyfbB.DoIt();

// Ejemplo para el puntero SUPER^
fbMyBase();
nBase := fbmyBase.nCnt;
fbMyFB_1();
nTHIS := fbMyFB_1.nCnt;

END_PROGRAM

// ---- 09_THIS_SUPER/THIS/FB_B.TcPOU
FUNCTION_BLOCK FB_B EXTENDS FB_A
VAR_INPUT
    nVarB : INT := 0;
END_VAR

nVarA := 11;
nVarB := 2;

METHOD DoIt : BOOL
VAR_INPUT
END_VAR
VAR
    nVarB : INT;
END_VAR
nVarB := 22; // Se establece la variable local nVarB.
THIS^.nVarB := 222; // La variable del bloque de funciones nVarB se establece aunque nVarB está oculta.
F_FunA(fbMyFbA := THIS^);  //F_FunA es llamado via THIS^.
END_METHOD

END_FUNCTION_BLOCK

// ---- 09_THIS_SUPER/THIS/FB_A.TcPOU
FUNCTION_BLOCK FB_A
VAR_INPUT
    nVarA: INT;
END_VAR

nVarA := 1;

END_FUNCTION_BLOCK

// ---- 09_THIS_SUPER/THIS/F_FunA.TcPOU
FUNCTION F_FunA : INT
VAR_INPUT
    fbMyFbA : FB_A;
END_VAR

END_FUNCTION

// ---- 09_THIS_SUPER/SUPER/FB_Base.TcPOU
FUNCTION_BLOCK FB_Base
VAR_OUTPUT
    nCnt : INT;
END_VAR

METHOD METH_DoAlso : BOOL
VAR_INPUT
END_VAR
METH_DoAlso := TRUE;
END_METHOD

METHOD METH_DoIt : BOOL
nCnt := -1;
END_METHOD

END_FUNCTION_BLOCK

// ---- 09_THIS_SUPER/SUPER/FB_1.TcPOU
FUNCTION_BLOCK FB_1 EXTENDS FB_Base
VAR_OUTPUT
    nBase: INT;
END_VAR

THIS^.METH_DoIt();      // llamada al metodo METH_DoIt del FB_1.
THIS^.METH_DoAlso();

SUPER^.METH_DoIt();     // llamada al metodo METH_DoIt del FB_Base.
SUPER^.METH_DoAlso();
nBase := SUPER^.nCnt;

METHOD METH_DoAlso : BOOL
nCnt := 123;    
METH_DoAlso := FALSE;
END_METHOD

METHOD METH_DoIt : BOOL
nCnt := 1111;    
METH_DoIt := TRUE;
END_METHOD

END_FUNCTION_BLOCK

// ---- 10_Interface/_10_Interface.TcPOU
PROGRAM _10_Interface
VAR
	//Ejemplo 1 Interface.
	Sensor 		: FB_Sensor;
	Calibrar 	: BOOL;
	Calibrado   : BOOL;
	Temperatura : REAL;
	Consigna    : REAL := 23.5;
	Valor       : INT;
	
	//Ejemplo 2 Interface.
	FB_A : FB_TestA;
	FB_B : FB_TestB;
	r32 :REAL;
	str1, str2: STRING;
	MyITF     : ITF_MyTest;
	r1, r2: REAL;
END_VAR

// Ejemplo 1 Interface.
IF Calibrar THEN
	Sensor.Calibrar();
ELSE
	Sensor.Descalibrar();
END_IF

Calibrado := Sensor.Calibrado;
Sensor.Consigna := Consigna;

Temperatura := Sensor.Temperatura;

Valor := Sensor.LeerValor();

// Ejemplo 2 Interface.
r32:= FB_A.METH3();

str1:= myFC(FB_A);
str2:= myFC(FB_B);

MyITF := FB_A;
r1 := MyITF.METH3();
MyITF := FB_B;
r2 := MyITF.METH3();

END_PROGRAM

// ---- 10_Interface/Interface1/FB_Sensor.TcPOU
FUNCTION_BLOCK FB_Sensor IMPLEMENTS I_Sensor
VAR_INPUT
END_VAR
VAR_OUTPUT
END_VAR
VAR
	_Calibrar 		: BOOL;
	Valor			: INT;
	_Temperatura 	: REAL;
	_Consigna       : REAL;

END_VAR

PROPERTY Calibrado : BOOL
GET
Calibrado := _Calibrar;
END_GET
END_PROPERTY


METHOD Calibrar
THIS^._Calibrar := TRUE;
END_METHOD

PROPERTY Consigna : REAL
SET
THIS^._Consigna := Consigna;
END_SET
END_PROPERTY

METHOD Descalibrar
THIS^._Calibrar := FALSE;
END_METHOD


METHOD LeerValor : INT
LeerValor := Valor;
END_METHOD


PROPERTY Temperatura : REAL
GET
Temperatura := THIS^._Temperatura;
END_GET
END_PROPERTY

END_FUNCTION_BLOCK

// ---- 10_Interface/Interface2/FB_TestA.TcPOU
FUNCTION_BLOCK FB_TestA IMPLEMENTS ITF_MyTest
VAR_INPUT
END_VAR
VAR_OUTPUT
END_VAR
VAR
	b1: BOOL;
	r32: REAL;
	str : STRING;
END_VAR

{warning 'Agregar implementación de método'}
METHOD METH1 : BOOL
METH1 := TRUE;
END_METHOD

{warning 'Agregar implementación de método'}
METHOD METH2 : STRING
METH2 := 'FB_TestA';
END_METHOD

{warning 'Agregar implementación de método'}
METHOD METH3 : REAL
METH3 := 3.14;
END_METHOD

{warning 'Agregar implementación de propiedad'}
PROPERTY Prop1 : BOOL
GET
Prop1:= b1;
END_GET
SET
b1 := Prop1;
END_SET
END_PROPERTY

{warning 'Agregar implementación de propiedad'}
PROPERTY Prop2 : REAL
GET
Prop2 := r32;
END_GET
SET
r32 := Prop2;
END_SET
END_PROPERTY

{warning 'Agregar implementación de propiedad'}
PROPERTY Prop3 : STRING
GET
Prop3 := str;
END_GET
SET
str := Prop3;
END_SET
END_PROPERTY

END_FUNCTION_BLOCK

// ---- 10_Interface/Interface2/FB_TestB.TcPOU
FUNCTION_BLOCK FB_TestB IMPLEMENTS ITF_MyTest
VAR_INPUT
END_VAR
VAR_OUTPUT
END_VAR
VAR
END_VAR

{warning 'Agregar implementación de método'}
METHOD METH1 : BOOL
END_METHOD

{warning 'Agregar implementación de método'}
METHOD METH2 : STRING
METH2 := 'FB_TestB';
END_METHOD

{warning 'Agregar implementación de método'}
METHOD METH3 : REAL
METH3 := 8.69;
END_METHOD

{warning 'Agregar implementación de propiedad'}
PROPERTY Prop1 : BOOL
GET
END_GET
SET
END_SET
END_PROPERTY

{warning 'Agregar implementación de propiedad'}
PROPERTY Prop2 : REAL
GET
END_GET
SET
END_SET
END_PROPERTY

{warning 'Agregar implementación de propiedad'}
PROPERTY Prop3 : STRING
GET
END_GET
SET
END_SET
END_PROPERTY

END_FUNCTION_BLOCK

// ---- 10_Interface/Interface2/myFC.TcPOU
FUNCTION myFC : STRING
VAR_INPUT
	myInterface : ITF_MyTest;
END_VAR
VAR
END_VAR

myFC := myInterface.METH2();

END_FUNCTION

// ---- 11_Puntero_y_Referencia/_11_Puntero_y_Referencia.TcPOU
PROGRAM _11_Puntero_y_Referencia
VAR
END_VAR


SR_Main_01();

SR_Main_02();

SR_Main_03();

SR_Main_04();

END_PROGRAM

// ---- 11_Puntero_y_Referencia/SR_Main_01.TcPOU
PROGRAM SR_Main_01
VAR
	inLocalAway : INT; // Variable integer local de SR_Main_01 para ser accedida externamente
END_VAR
	
VAR
    aR20: ARRAY[1..20] OF REAL; //Declara un array de 20 elementos del tipo REAL.
    inIndex: INT; //Declara la variable de indice del array para el acceso indirecto
    xNewVal: BOOL; //Indica que hay una nueva lectura del sensor de fuerza.
    rFuerza: REAL; //Valor de fuerza del sensor.
END_VAR

VAR 
    stRectangulo1 : st_Rectangulo; // Estructura que contiene los datos del rectangulo1 A, B y su area
    stRectangulo2 : st_Rectangulo; // Estructura que contiene los datos del rectangulo2 A, B y su area
    stRectangulo3 : st_Rectangulo; // Estructura que contiene los datos del rectangulo3 A, B y su area

    refRectangulo : REFERENCE TO st_Rectangulo := stRectangulo3; // Hace Referencia a stRectangulo3   
END_VAR

// Ejemplo01: Se asigna valores del 1 al 20 a cada elemento del array mediante un bucle.
FOR inIndex:=1 TO 20 BY 1 DO  // Se empieza por el valor de la variable indice a 1, hasta 20
    aR20[inIndex] := inIndex; // Al elemento aR20[inIndex] se le asigna el valor de inIndex
END_FOR;                      // Se incrementa inIndex y se repite el proceso.

// Ejemplo02: Creamos un FIFO en el que guardamos un valor analógico de fuera a cada impulso de la señal xNewVal.
IF xNewVal THEN                // Si hay un nuevo valor de fuerza realizamos el codigo.
    xNewVal := FALSE;          // Reset de la señal xNewVal.

    FOR inIndex:=20 TO 2 BY -1 DO // Variable indice a 20, hasta 2.
        aR20[inIndex] := aR20[inIndex-1]; //Desplazamiento de los valores en el FIFO --->
    END_FOR;                             // Se decrementa inIndex y se repite el proceso.

    aR20[1] := rFuerza; // Entrada del valor de fuerza en el primer elemento del FIFO.
END_IF

//*********************************************************************************************************

// Asignación de valores a los lados de los tres rectángulos.

// Asignación de valores de los lados del rectángulo 1
stRectangulo1.rAside := 44; //Valor del lado A.
stRectangulo1.rBside := 32; //Valor del lado B.

// Asignación de valores de los lados del rectángulo 2
stRectangulo2.rAside := 12.8; //Valor del lado A.
stRectangulo2.rBside := 320.4; //Valor del lado B.

// Asignación de valores de los lados del rectángulo 3
stRectangulo3.rAside := 1024.2; //Valor del lado A.
stRectangulo3.rBside := 2048.4; //Valor del lado B.

// Cálculo del área del rectángulo pasando valores a la función
stRectangulo1.rArea := Fc_AreaCalcVal(i_rAside:=stRectangulo1.rAside, i_rBside:= stRectangulo1.rBside);

// Cálculo del área del rectángulo pasando un puntero a la función
Fc_AreaCalcPoint(ADR(stRectangulo2));

// Cálculo del área del rectángulo pasando una referencia a la función
Fc_AreaCalcRef(refRectangulo);

END_PROGRAM

// ---- 11_Puntero_y_Referencia/Fc_AreaCalcVal.TcPOU
FUNCTION Fc_AreaCalcVal : REAL
VAR_INPUT
    i_rASide    : REAL; // Parámetro de entrada que contiene el lado A del rectangulo.
    i_rBSide    : REAL; // Parámetro de entrada que contiene el lado B del rectangulo.
END_VAR

Fc_AreaCalcVal := i_rASide * i_rBSide; // Retorna el resultado de multiplicar el lado A por el lado B.

END_FUNCTION

// ---- 11_Puntero_y_Referencia/Fc_AreaCalcPoint.TcPOU
FUNCTION Fc_AreaCalcPoint : REAL
VAR_INPUT
    i_ptstRect : POINTER TO st_Rectangulo; // Puntero de entrada con la dirección de la estructura.
END_VAR

// El valor del area, de la estructura indicada por la dirección del puntero es igual al
// valor del lado A de la estructura indicada por la dirección del puntero por
// el valor del lado B de la estructura indicada por la dirección del puntero
i_ptstRect^.rArea := i_ptstRect^.rASide * i_ptstRect^.rBSide;

END_FUNCTION

// ---- 11_Puntero_y_Referencia/Fc_AreaCalcRef.TcPOU
FUNCTION Fc_AreaCalcRef : REAL
VAR_INPUT
    i_Ref : REFERENCE TO st_Rectangulo;
END_VAR

i_Ref.rArea := i_Ref.rASide * i_Ref.rBSide;

END_FUNCTION

// ---- 11_Puntero_y_Referencia/SR_Main_02.TcPOU
PROGRAM SR_Main_02
VAR
    in01    : INT; //Declaración de la variable in01 de tipo entero.
    in02    : INT := 123; //Declaración e inicialización de la variable in02 de tipo entero.
    in03    : INT; //Declaración de la variable in03 de tipo entero.

    pint    : POINTER TO INT; //Declaración de un puntero para acceder a variables del tipo entero.
END_VAR

// Ejemplo de uso básico de los operadores ADR y del operador de contenido ^
// Se muestra como asignar a un puntero la dirección de memoria de una variable y como leer/escribir
// así como un ejemplo de acceso a variables locales de otros programas.

pint := ADR(in01); //Asignamos al puntero la dirección de memoria donde se ubica la variable in01.
pint^ := 44;     //A la posición de memoria indicada por el puntero, le asignamos el valor 44
                 //Por tanto a la variable in01 se le ha escrito el valor 44.

in02 := in01; // in02 será igual a 44.

pint := ADR(in02); //Cambiamos la dirección para acceder a la dirección de la variable in02.
in03 := pint^; // in03 tomara el valor del contenido de la posición de memoria contenida en el
               // que hemos asignado la dirección de in02, por tanto in03= 123.

pint := ADR(SR_Main_01.inLocalAway); //Cargamos la dirección de memoria de una variable local de 
                                     // otro programa, la que sería inaccesible por otros medios.
pint^ := 240 ; // La varible local del programa SR_Main_01.inLocalAway tomará el valor 240

END_PROGRAM

// ---- 11_Puntero_y_Referencia/SR_Main_03.TcPOU
PROGRAM SR_Main_03
VAR
    stMotor_01 : stMotorCtrl; // Estructura de control del motor 1
    stMotor_02 : stMotorCtrl; // Estructura de control del motor 2
    stMotor_03 : stMotorCtrl; // Estructura de control del motor 3
    pstMotorCtrl : POINTER TO stMotorCtrl; // Puntero para acceder a estructuras del tipo stMotorCtrl.
    xMarcha : BOOL; // Pulsador marcha motores.
END_VAR

VAR
    aintFIFO    : ARRAY[1..20] OF INT; // Array de 20 enteros.
    aintFIFO2   : ARRAY[1..20] OF INT; // Array de 20 enteros.
    paint       : POINTER TO ARRAY[1..20] OF INT; // Puntero al array.
    pint        : POINTER TO INT; // Puntero a un entero.
END_VAR

// Ejemplo básico de como acceder a estructuras de datos mediante punteros.
// La estructura de datos empleada es una llamada a stMotorCtrl, que coincide un bit de marcha, otro de paro y
// valores de velocidad en Rpms y tiempo de aceleración/deceleración.

// Asignamos valores a la estructura para el control del motor 1.

stMotor_01.rTpoAcelDecel := 5.4; // Tiempo para acelerar/decelerar hasta alcanazar la velocidad.
stMotor_01.rVelRpm := 1436.2; // Velocidad en RPM.
stMotor_01.xMotorOff := TRUE; // Bit de paro ON.
stMotor_01.xMotorOn := FALSE   ; // Bit de marcha OFF.

pstMotorCtrl := ADR(stMotor_01); // Cargamos la dirección de memoria de la estructura del motor 1
stMotor_02 := pstMotorCtrl^; // Copia el contenido de la zona de memoria apuntada a la
                             // estructura del motor 2, en este caso el resultado es el mismo
                             // que se obtendría con stMotor_02:= stMotor_01;

stMotor_03 := stMotor_02; // Copia los mismos valores al motor 3;

IF xMarcha THEN         // Si se pulsa marcha máquina
    pstMotorCtrl^.xMotorOn := TRUE; // Se activa el bit de marcha al que apunta el puntero (stMotor_01).
    pstMotorCtrl^.xMotorOff := FALSE; // Se desactiva el bit de paro al que apunta el puntero (stMotor_01)
END_IF

//***************************************************************************************************************
// Ejemplo basico de como acceder a arrays mediante punteros:
paint := ADR(aintFIFO); // _Asignamos la dirección del array al puntero.
paint^[3] := 4; // Dentro del array podemos acceder a un elemento en concreto
aintFIFO2 := paint^; // O copiar el array apuntado entero, sobre otro array
pint := paint + (4 * SIZEOF (INT)); // Tambien se puede crear un puntero a un INT para acceder a uno de los
                                    // elementos del array. Tomamos la dirección inicial del array y le
                                    // sumampos un offeset de tantos bytes como se necesitan para el tipo de 
                                    // datos INT y lo multiplicamos por el indice del array al que queremos
                                    // acceder. SIZEOF (TYPE) retorna el número de bytes según el tipo de datos.

pint^ := 5;                         // Asignamos el valor de 5, aintFIFO[5]:=5 sería lo mismo.

END_PROGRAM

// ---- 11_Puntero_y_Referencia/SR_Main_04.TcPOU
PROGRAM SR_Main_04
VAR
 arFIFO  : ARRAY[1..20] OF REAL; // FIFO con los valores de fuerza registrados.
 intIdx  : INT;                  // Variable de indice.
 rIncAng : REAL;                 // Valor de incremento angular para generación de senoide.
 rValAng : REAL;                 // Valor actual de angulo.
 rValSin : REAL;                 // Amplitud de la senoide superpuesta.
 rVMed   : REAL;                 // Resultado del cálculo.

 refFIFO : REFERENCE TO ARRAY[1..20] OF REAL := arFIFO; // Crea una referencia y la asigna a arFIFO
 rMedRef : REAL;           // Resultado del cálculo para el ejemplo de pase de valores por Ref.
END_VAR

// Ejemplo de como realizar el cálculo del valor medio de las lecturas de fuerza contenidas en arFIFO
// mediante la función Fc_AverageValues (Pase de parámetros por valores) y Fc_AverageReferencia (Pase de
// parámetros por referencia)
// Lo que se pretende es ver las ventajas del pase por referencia

// Asignación de valores para llenar el FIFO a efectos de tener algunos valores para el cálculo de la media
// al valor 124 le superpone una variación senoidal de amplitud 6

rIncAng := (2 * 3.14159) / 20.0; // 2 * PI Radianes dividido entre 20 puntos.
rValAng := 0.0;                   // Valor inicial del angulo.

FOR intIdx :=1 TO 20 BY 1 DO
 rValSin := SIN(rValAng) * 6;         // Valor del seno para una amplitud de 6
 arFIFO[intIdx] := 124.0 + rValSin;  // A un nivel de 124.0 se superpone un seno de amplitud 6.
 rValAng := rValAng + rIncAng;       // Próximo valor angular. 
END_FOR;

// Con el FIFO de valores llamaremos a la función para el cálculo de la media pasando valores.
// Lo que no sería para nada adecuado por tratarse de muchos parámetros.

rVMed:= Fc_AverageValues( i_REALV1  := arFIFO[1],
                          i_REALV2  := arFIFO[2],
                          i_REALV3  := arFIFO[3],
                          i_REALV4  := arFIFO[4], 
                          i_REALV5  := arFIFO[5],
                          i_REALV6  := arFIFO[6], 
                          i_REALV7  := arFIFO[7],
                          i_REALV8  := arFIFO[8],
                          i_REALV9  := arFIFO[9],
                          i_REALV10 := arFIFO[10],
                          i_REALV11 := arFIFO[11],
                          i_REALV12 := arFIFO[12],
                          i_REALV13 := arFIFO[13],
                          i_REALV14 := arFIFO[14],
                          i_REALV15 := arFIFO[15],
                          i_REALV16 := arFIFO[16],
                          i_REALV17 := arFIFO[17],
                          i_REALV18 := arFIFO[18],
                          i_REALV19 := arFIFO[19],
                          i_REALV20 := arFIFO[20]);

// Con el FIFO lleno de valores llamaremos a la función para el cálculo de la media pasando valores por referencia
// para ver lo sencillo que resulta en este caso.

rMedRef := Fc_AverageReferencia(i_Ref:=refFIFO);

END_PROGRAM

// ---- 11_Puntero_y_Referencia/Fc_AverageValues.TcPOU
FUNCTION Fc_AverageValues : REAL
VAR_INPUT
    i_REALV1  : REAL; //Valor posición 1
    i_REALV2  : REAL; //Valor posición 2
    i_REALV3  : REAL; //Valor posición 3
    i_REALV4  : REAL; //Valor posición 4
    i_REALV5  : REAL; //Valor posición 5
    i_REALV6  : REAL; //Valor posición 6
    i_REALV7  : REAL; //Valor posición 7
    i_REALV8  : REAL; //Valor posición 8
    i_REALV9  : REAL; //Valor posición 9
    i_REALV10 : REAL; //Valor posición 10
    i_REALV11 : REAL; //Valor posición 11
    i_REALV12 : REAL; //Valor posición 12
    i_REALV13 : REAL; //Valor posición 13
    i_REALV14 : REAL; //Valor posición 14
    i_REALV15 : REAL; //Valor posición 15
    i_REALV16 : REAL; //Valor posición 16
    i_REALV17 : REAL; //Valor posición 17
    i_REALV18 : REAL; //Valor posición 18
    i_REALV19 : REAL; //Valor posición 19
    i_REALV20 : REAL; //Valor posición 20
END_VAR

//Retorna la suma de todos los valores dividida del número de valores que son 20.

Fc_AverageValues := (i_REALV1 + i_REALV2 + i_REALV3 + i_REALV4 + i_REALV5 + i_REALV6 + i_REALV7 + 
                    i_REALV8 + i_REALV9 + i_REALV10 + i_REALV11 + i_REALV12 + i_REALV13 + 
                    i_REALV14 + i_REALV15 + i_REALV16 + i_REALV17 + i_REALV18 + 
                    i_REALV19 + i_REALV20) / 20.0 ;

END_FUNCTION

// ---- 11_Puntero_y_Referencia/Fc_AverageReferencia.TcPOU
FUNCTION Fc_AverageReferencia : REAL
VAR_INPUT
 i_Ref : REFERENCE TO ARRAY[1..20] OF REAL;
END_VAR
VAR
 intIdx : INT;      // Variable indice para el bucle.
 rVAcum : REAL:=0; // Valor acumulado.
END_VAR

// Retorna la suma de todos los valores divida del número de valores que son 20.

FOR intIdx:=1 TO 20 BY 1 DO
 rVAcum := rVAcum + i_Ref[intIdx];
END_FOR;
Fc_AverageReferencia := rVAcum / 20.0;

END_FUNCTION

// ---- 12_Concepto Keyword Abstract/_12_Concepto_Keyword_Abstract.TcPOU
PROGRAM _12_Concepto_Keyword_Abstract
VAR
 	fbLoadCell:REFERENCE TO AbstractLoadCell;
	   
	ConcreteCSVLogger:ConcreteCSVLogger;
    ConcreteAdsLogger:ConcreteADSLogger;
	AbstractLogger:POINTER TO AbstractLogger;
 
    LogNow:BOOL;
    Process1:INT;
    Process2:INT;
END_VAR

(*
Concepto ABSTRACTO
La palabra clave ABSTRACT está disponible para bloques de funciones, métodos y propiedades. Permite la implementación de un proyecto PLC con niveles de abstracción.
La abstracción es un concepto clave de la programación orientada a objetos. Los diferentes niveles de abstracción contienen aspectos de implementación generales o específicos.

CONCEPTO ABSTRACTO 1:	
Disponible en TC3.1 Build 4024

Aplicación de la abstracción
Es útil implementar funciones básicas o puntos en común de diferentes clases en una clase básica abstracta. Se implementan aspectos específicos en subclases no abstractas.
El principio es similar al uso de una interfaz. Las interfaces corresponden a clases puramente abstractas que contienen sólo métodos y propiedades abstractas.
Una clase abstracta también puede contener métodos y propiedades no abstractos.

Reglas para el uso de la palabra clave ABSTRACT
Los bloques de funciones abstractas no se pueden instanciar.
Los bloques de funciones abstractas pueden contener métodos y propiedades abstractos y no abstractos.
Los métodos abstractos o las propiedades no contienen ninguna implementación (solo la declaración).
Si un bloque de funciones contiene un método o propiedad abstracta, debe ser abstracta.
Los bloques de funciones abstractas deben extenderse para poder implementar los métodos o propiedades abstractas.
Por lo tanto: Un FB derivado debe implementar los métodos / propiedades de su FB básico o también debe definirse como abstracto.
Muestra
Clase básica abstracta:

FUNCTION_BLOCK ABSTRACT FB_System_Base
Los puntos en común de todos los módulos del sistema se implementan en esta clase básica abstracta. Contiene la propiedad no abstracta "nSystemID" y el método abstracto "Execute" para esto:

PROPERTY nSystemID : UINT
METHOD ABSTRACT Execute
mientras que la implementación de "nSystemID" es la misma para todos los sistemas, la implementación del método "Execute" difiere para los sistemas individuales.

Subclase no abstracta:

FUNCTION_BLOCK FB_StackSystem EXTENDS FB_System_Base
Las clases no abstractas que se derivan de la clase básica se implementan para los sistemas específicos. Esta subclase representa una pila. Dado que no es abstracto, debe implementar el método "Execute" que define la ejecución específica de la pila:

METHOD Execute

*)

// Process 1 assigns a logger and starts task 2.
CASE Process1 OF
    0: IF LogNow THEN
            LogNow:=FALSE;
            AbstractLogger:= ADR(ConcreteAdsLogger);
            Process2 :=1;
            Process1:=Process1+1;               
        END_IF
     
    1: IF Process2 = 0 THEN
            AbstractLogger:= ADR(ConcreteCSVLogger);
            Process2:=1;
            Process1:=Process1+1;   
       END_IF
        
     2:IF Process2 = 0 THEN
            AbstractLogger:= ADR(ConcreteAdsLogger);
            Process2:=1;
            Process1:=Process1+1;   
       END_IF
        
      3: IF Process2 = 0 THEN
            AbstractLogger:= ADR(ConcreteCSVLogger);
            Process2:=1;
            Process1:=Process1+1;   
       END_IF
        
      4:IF Process2 = 0 THEN
            Process1:=0;    
       END_IF
END_CASE
 
//Process 2 does its task indepently of the assigned type of logger. 
CASE process2 OF
    1: AbstractLogger^.LogMessage(CONCAT('Important message ',INT_TO_STRING(Process1)));
       process2:=process2+1;                
         
    2: AbstractLogger^();
       IF NOT AbstractLogger^.Busy THEN
            process2:=0;    
       END_IF
END_CASE

END_PROGRAM

// ---- 12_Concepto Keyword Abstract/AbstractLoadCell.TcPOU
FUNCTION_BLOCK ABSTRACT AbstractLoadCell
VAR_INPUT
END_VAR
VAR_OUTPUT
END_VAR
VAR
END_VAR

METHOD PUBLIC ABSTRACT GetActualValue : LREAL
VAR_INPUT
END_VAR
END_METHOD

END_FUNCTION_BLOCK

// ---- 12_Concepto Keyword Abstract/ConcreteCSVLogger.TcPOU
{attribute 'hide_all_locals'}
FUNCTION_BLOCK FINAL ConcreteCSVLogger EXTENDS AbstractLogger
VAR
    fbFileOpen:FB_FileOpen;
    fbFilePuts:FB_FilePuts;
    fbFileClose:FB_FileClose;
    State:INT;
    Message:STRING;
END_VAR

CASE State OF
    0:  IF _Busy THEN
            State:=State+1;
        END_IF
     
    1:  fbFileOpen(bExecute:=FALSE);
        fbFileOpen(sNetId:='', //'xxx.xx.xxx.1.1.1',
            sPathName:='C:\Log.csv',
            nMode:=FOPEN_MODEAPPEND,
            bExecute:=TRUE);
        State:=State+1;
         
    2:  fbFileOpen(bExecute:=FALSE);
        IF NOT fbFileOpen.bBusy THEN
            State:=State+1;
        END_IF
     
    3:  fbFilePuts(bExecute :=FALSE);
        fbFilePuts( bExecute:=TRUE,
                    sNetId:='',//'xxx.xx.xxx.1.1.1',
                    hFile:=fbFileOpen.hFile,
                    sLine:=Message);
        State:=State+1;
     
    4:  fbFilePuts(bExecute:=FALSE);
        IF NOT fbFilePuts.bBusy THEN
            State:=State+1;
        END_IF
         
    5:  fbFileClose(bExecute :=FALSE);
        fbFileClose(sNetId:='',//'xxx.xx.xxx.1.1.1',
                    bExecute:=TRUE,
                    hFile:= fbFileOpen.hFile);
        State:=State+1; 
         
    6:  fbFileClose(bExecute:=FALSE);
        IF NOT fbFileClose.bBusy THEN
            State:=0;
            _Busy:=FALSE;
        END_IF
END_CASE

METHOD PROTECTED  InternalLog
VAR_INPUT
    Message:STRING;
END_VAR
THIS^.Message:=CONCAT(Message,'$n');
_Busy:=TRUE;
END_METHOD

END_FUNCTION_BLOCK

// ---- 12_Concepto Keyword Abstract/AbstractLogger.TcPOU
FUNCTION_BLOCK ABSTRACT AbstractLogger

VAR
	_Busy:BOOL; //Backing variable for Busy property.
END_VAR

{attribute 'monitoring' := 'variable'}
PROPERTY Busy : BOOL
GET
Busy:=_Busy;
END_GET
SET
END_SET
END_PROPERTY

METHOD PROTECTED ABSTRACT InternalLog
VAR_INPUT
	Message:STRING;
END_VAR
END_METHOD

METHOD PUBLIC LogMessage
VAR_INPUT
	Message:STRING;
END_VAR
VAR
    GetSystemTime : NT_GetTime:=(NetID:=''); //'xxx.xxx.xxx.1.1.1');
END_VAR
// Retrieve a the current system time and combine it with the input message. 
GetSystemTime(START:=FALSE);
REPEAT
    GetSystemTime(START:=TRUE);
UNTIL (NOT GetSystemTime.BUSY)
END_REPEAT
 
//Call abstract method
InternalLog(Message:=CONCAT(CONCAT(Message,', '),SYSTEMTIME_TO_STRING(GetSystemTime.TIMESTR)));
END_METHOD

END_FUNCTION_BLOCK

// ---- 12_Concepto Keyword Abstract/ConcreteADSLogger.TcPOU
FUNCTION_BLOCK PUBLIC FINAL ConcreteADSLogger EXTENDS AbstractLogger
VAR_INPUT
END_VAR
VAR_OUTPUT
END_VAR
VAR
END_VAR

METHOD PROTECTED InternalLog
VAR_INPUT
     Message:STRING;
END_VAR
_Busy:=TRUE;
 
ADSLOGSTR(    msgCtrlMask:=ADSLOG_MSGTYPE_LOG,
              msgFmtStr:=Message,
              strArg:='');
             
_Busy:=FALSE;
END_METHOD

END_FUNCTION_BLOCK

// ---- 13_FB_Abstracto_vs_Interface/1_FB_Abstracto/_13_1_Main_Abstract.TcPOU
PROGRAM _13_1_Main_Abstract
VAR	
	fbFullTimeEmployee	:	FB_FullTimeEmployee;
	fbContractEmployee	:	FB_ContractEmployee;
	refEmployee			:	REFERENCE TO FB_Employee;
	aFullName			:	ARRAY[1..2] OF STRING;
	aMonthlySalary		:	ARRAY[1..2] OF LREAL;
END_VAR

fbFullTimeEmployee.nPersonnelNumber := 1;
fbFullTimeEmployee.sFirstName := 'John';
fbFullTimeEmployee.sLastName := 'Taylor';
fbFullTimeEmployee.nAnnualSalary := 60000;
// access via concrete FB
aFullName[1] := fbFullTimeEmployee.GetFullName();
aMonthlySalary[1] := fbFullTimeEmployee.GetMonthlySalary();
// access via abstract FB
refEmployee REF= fbFullTimeEmployee;
aFullName[1] := refEmployee.GetFullName();
aMonthlySalary[1] := refEmployee.GetMonthlySalary();

fbContractEmployee.nPersonnelNumber := 2;
fbContractEmployee.sFirstName := 'Tim';
fbContractEmployee.sLastName := 'Brown';
fbContractEmployee.nMonthlyHours := 160;
fbContractEmployee.nHourlyPay := 35;
// access via concrete FB
aFullName[2] := fbContractEmployee.GetFullName();
aMonthlySalary[2] := fbContractEmployee.GetMonthlySalary();
// access via abstract FB
refEmployee REF= fbContractEmployee;
aFullName[2] := refEmployee.GetFullName();
aMonthlySalary[2] := refEmployee.GetMonthlySalary();

END_PROGRAM

// ---- 13_FB_Abstracto_vs_Interface/1_FB_Abstracto/FB_FullTimeEmployee.TcPOU
{attribute 'hide_all_locals'}
FUNCTION_BLOCK PUBLIC FB_FullTimeEmployee EXTENDS FB_Employee
VAR_INPUT
END_VAR
VAR_OUTPUT
END_VAR
VAR
	nAnnualSalaryBacking	:	UINT;
END_VAR

METHOD PUBLIC GetMonthlySalary : LREAL
VAR_INPUT
END_VAR
GetMonthlySalary := nAnnualSalary / 12;
END_METHOD

{attribute 'monitoring' := 'variable'}
PROPERTY PUBLIC nAnnualSalary : UINT
GET
nAnnualSalary := nAnnualSalaryBacking;
END_GET
SET
nAnnualSalaryBacking := nAnnualSalary;
END_SET
END_PROPERTY

END_FUNCTION_BLOCK

// ---- 13_FB_Abstracto_vs_Interface/2_Interfaz/_13_2_Main_Interfaz.TcPOU
PROGRAM _13_2_Main_Interfaz
VAR
	fbFullTimeEmployee	:	FB_FullTimeEmployee_1;
	fbContractEmployee	:	FB_ContractEmployee_1;
	ipEmployee			:	I_Employee;
	aFullName			:	ARRAY[1..2] OF STRING;
	aMonthlySalary		:	ARRAY[1..2] OF LREAL;
END_VAR

fbFullTimeEmployee.nPersonnelNumber := 1;
fbFullTimeEmployee.sFirstName := 'John';
fbFullTimeEmployee.sLastName := 'Taylor';
fbFullTimeEmployee.nAnnualSalary := 60000;
// access via FB
aFullName[1] := fbFullTimeEmployee.GetFullName();
aMonthlySalary[1] := fbFullTimeEmployee.GetMonthlySalary();
// access via interface
ipEmployee := fbFullTimeEmployee;
aFullName[1] := ipEmployee.GetFullName();
aMonthlySalary[1] := ipEmployee.GetMonthlySalary();

fbContractEmployee.nPersonnelNumber := 2;
fbContractEmployee.sFirstName := 'Tim';
fbContractEmployee.sLastName := 'Brown';
fbContractEmployee.nMonthlyHours := 160;
fbContractEmployee.nHourlyPay := 35;
// access via FB
aFullName[2] := fbContractEmployee.GetFullName();
aMonthlySalary[2] := fbContractEmployee.GetMonthlySalary();
// access via interface
ipEmployee := fbContractEmployee;
aFullName[2] := ipEmployee.GetFullName();
aMonthlySalary[2] := ipEmployee.GetMonthlySalary();

END_PROGRAM

// ---- 13_FB_Abstracto_vs_Interface/3_Combinacion/_13_3_Main_Combinacion.TcPOU
PROGRAM _13_3_Main_Combinacion
VAR
	fbFullTimeEmployee	:	FB_FullTimeEmployee_2;
	fbContractEmployee	:	FB_ContractEmployee_2;
	refEmployee			:	REFERENCE TO FB_Employee_1;
	ipEmployee			:	I_Employee_1;	
	aFullName			:	ARRAY[1..2] OF STRING;
	aMonthlySalary		:	ARRAY[1..2] OF LREAL;
END_VAR

fbFullTimeEmployee.nPersonnelNumber := 1;
fbFullTimeEmployee.sFirstName := 'John';
fbFullTimeEmployee.sLastName := 'Taylor';
fbFullTimeEmployee.nAnnualSalary := 60000;
// access via concrete FB
aFullName[1] := fbFullTimeEmployee.GetFullName();
aMonthlySalary[1] := fbFullTimeEmployee.GetMonthlySalary();
// access via abstract FB
refEmployee REF= fbFullTimeEmployee;
aFullName[1] := refEmployee.GetFullName();
aMonthlySalary[1] := refEmployee.GetMonthlySalary();
// access via interface
ipEmployee := fbFullTimeEmployee;
aFullName[1] := ipEmployee.GetFullName();
aMonthlySalary[1] := ipEmployee.GetMonthlySalary();

fbContractEmployee.nPersonnelNumber := 2;
fbContractEmployee.sFirstName := 'Tim';
fbContractEmployee.sLastName := 'Brown';
fbContractEmployee.nMonthlyHours := 160;
fbContractEmployee.nHourlyPay := 35;
// access via concrete FB
aFullName[2] := fbContractEmployee.GetFullName();
aMonthlySalary[2] := fbContractEmployee.GetMonthlySalary();
// access via abstract FB
refEmployee REF= fbContractEmployee;
aFullName[2] := refEmployee.GetFullName();
aMonthlySalary[2] := refEmployee.GetMonthlySalary();
// access via interface
ipEmployee := fbContractEmployee;
aFullName[2] := ipEmployee.GetFullName();
aMonthlySalary[2] := ipEmployee.GetMonthlySalary();

END_PROGRAM

// ---- 13_FB_Abstracto_vs_Interface/3_Combinacion/FB_ContractEmployee_2.TcPOU
{attribute 'hide_all_locals'}
FUNCTION_BLOCK PUBLIC FB_ContractEmployee_2 EXTENDS FB_Employee_1
VAR_INPUT
END_VAR
VAR_OUTPUT
END_VAR
VAR
	nHourlyPayBacking		:	UINT;
	nMonthlyHoursBacking	:	UINT;
END_VAR

METHOD PUBLIC GetMonthlySalary : LREAL
VAR_INPUT
END_VAR
GetMonthlySalary := nMonthlyHours * nHourlyPay;
END_METHOD

{attribute 'monitoring' := 'variable'}
PROPERTY PUBLIC nHourlyPay : UINT
GET
nHourlyPay := nHourlyPayBacking;
END_GET
SET
nHourlyPayBacking := nHourlyPay;
END_SET
END_PROPERTY

{attribute 'monitoring' := 'variable'}
PROPERTY PUBLIC nMonthlyHours : UINT
GET
nMonthlyHours := nMonthlyHoursBacking;
END_GET
SET
nMonthlyHoursBacking := nMonthlyHours;
END_SET
END_PROPERTY

END_FUNCTION_BLOCK

// ---- 14_Interface_Fluida/_14_Interface_Fluida.TcPOU
PROGRAM _14_Interface_Fluida
VAR
	fMyResult1 : LREAL;
	fbCalculate : FB_Calculate;
	
	fMyResult2 : LREAL;
	fbCalcul : FB_Calcul;
END_VAR

// 14_1 : se ha realizado un ejemplo de interface fluida.
fMyResult1 := fbCalculate.Clear()
		            		.SetNumber(12)
		        			.DecreaseBy(2)
		        			.IncreaseBy(3.9)
	                		.MultiplyBy(5)
		        			.DivideBy(3)
		        			.GetResult();							
													
						
// 14_2 : se ha optimazado un poco, para que la interfaz fluida no deje ir encadenando metodos que se contradigan entre si...	
// por ejemplo el metodo SetNumber() solo tiene sentido después del metodo Clear()..
// y los metodos de realizar operaciones solo tienen sentido si ha realizado antes el metodo SetNumber()...					
fMyResult2 := fbCalcul.Clear()
						.SetNumber(12)
						.DecreaseBy(2)
		        		.IncreaseBy(3.9)
	                	.MultiplyBy(5)
		        		.DivideBy(3)						
						.GetResult();											

// 14_3 : la forma mas optima sería que primero de todo solo pidiese el metodo Clear()
// y despues solo saliese el metodo SetNumber() 
// y después ya se pudiesen poner solo los metodos de operaciones y el de GetResult()

END_PROGRAM

// ---- 14_Interface_Fluida/14_1/FB_Calculate.TcPOU
FUNCTION_BLOCK FB_Calculate IMPLEMENTS I_Calculate
VAR
	{attribute  'hide'}
	lResult : LREAL := 0;
END_VAR


METHOD Clear : I_Calculate
MEMSET(destAddr:= ADR(lResult),fillByte :=0, n:=SIZEOF(lResult));
Clear := THIS^;
END_METHOD


METHOD DecreaseBy : I_Calculate
VAR_INPUT
	lDecreaseBy : REAL;
END_VAR
lResult := lResult - lDecreaseBy;
DecreaseBy := THIS^;
END_METHOD


METHOD DivideBy : I_Calculate
VAR_INPUT
	lDivideBy : REAL;
END_VAR
IF lDivideBy = 0 THEN
	lResult := 0;
ELSE	
	lResult := lResult / lDivideBy;
END_IF

DivideBy := THIS^;
END_METHOD


METHOD GetResult : LREAL
GetResult := lResult;
END_METHOD

METHOD IncreaseBy : I_Calculate
VAR_INPUT
	lIncreaseBy : REAL;
END_VAR
lResult := lResult + lIncreaseBy;
IncreaseBy := THIS^;
END_METHOD


METHOD MultiplyBy : I_Calculate
VAR_INPUT
	lMultiplyBy : REAL;
END_VAR
lResult := lResult * lMultiplyBy;
MultiplyBy := THIS^;
END_METHOD

METHOD SetNumber : I_Calculate
VAR_INPUT
	lNumber : LREAL;
END_VAR
lResult := lNumber;
SetNumber := THIS^;
END_METHOD

END_FUNCTION_BLOCK

// ---- 14_Interface_Fluida/14_2/FB_Calcul.TcPOU
FUNCTION_BLOCK FB_Calcul IMPLEMENTS I_Clear, I_SetNumber, I_Operation

VAR
	{attribute  'hide'}
	lResult : LREAL := 0;
END_VAR


METHOD Clear : I_SetNumber
MEMSET(destAddr:= ADR(lResult),fillByte :=0, n:=SIZEOF(lResult));
Clear := THIS^;
END_METHOD


METHOD DecreaseBy : I_Operation
VAR_INPUT
	lDecreaseBy	: REAL;
END_VAR
lResult := lResult - lDecreaseBy;
DecreaseBy := THIS^;
END_METHOD

{warning 'Agregar implementación de método'}
METHOD DivideBy : I_Operation
VAR_INPUT
	lDivideBy	: REAL;
END_VAR
IF lDivideBy = 0 THEN
	lResult := 0;
ELSE	
	lResult := lResult / lDivideBy;
END_IF

DivideBy := THIS^;
END_METHOD


METHOD GetResult : LREAL
GetResult := lResult;
END_METHOD


METHOD IncreaseBy : I_Operation
VAR_INPUT
	lIncreaseBy	: REAL;
END_VAR
lResult := lResult + lIncreaseBy;
IncreaseBy := THIS^;
END_METHOD


METHOD MultiplyBy : I_Operation
VAR_INPUT
	lMultiplyBy	: REAL;
END_VAR
lResult := lResult * lMultiplyBy;
MultiplyBy := THIS^;
END_METHOD


METHOD SetNumber : I_Operation
VAR_INPUT
	lNumber	: LREAL;
END_VAR
lResult := lNumber;
SetNumber := THIS^;
END_METHOD

END_FUNCTION_BLOCK

// ---- 15_Interface_vs_Herencia/_15_Interface_vs_Herencia.TcPOU
PROGRAM _15_Interface_vs_Herencia
VAR
	//Nivel Sensor: 
	fbNivelSensor			: FB_NivelSensor;
	nNivelAnalogSensor 		: INT := 8000;
	nScaledNivelSensor 		: INT;
	nSensorNivelMaxValue 	: INT;

	//UltraSonidos
	fbUltraSonic 			: FB_UltraSonicSensor;
	nAnalogSensor 			: INT := 8000;
	nScaledSensor 			: INT;
	nSensorMaxValue 		: INT;
	
	//Variador de Frequencia
	fbVFD1 					: FB_VFD;
	bCoil1 					: BOOL;
	nFreqIn1  				: INT := 25;
	nFreqOut1 				: INT;	
	bStartVFD1 				: BOOL;
	
	//Pump
	fbPump1 				: FB_Pump;
	bCoilPump1				: BOOL;
	nFreqInPump1  			: INT := 25;
	nFreqOutPump1 			: INT;	
	bStartPump1 			: BOOL;	
END_VAR

//Nivel Sensor
fbNivelSensor.AnalogSignal := nNivelAnalogSensor;
fbNivelSensor.MaxValue := 6;
nScaledNivelSensor := fbNivelSensor.ScaledAnalog;
fbNivelSensor.Scale();

//UltraSonidos
fbUltraSonic.AnalogSignal := nAnalogSensor;
fbUltraSonic.MaxValue := 6;
nScaledSensor := fbUltraSonic.ScaledAnalog;
fbUltraSonic.Scale();

//Variador de Frequencia
fbVFD1.AnalogSignal := nFreqIn1;
bCoil1 := fbVFD1.Coil;
nFreqOut1 := fbVFD1.ScaledAnalog;
fbVFD1.Scale();

IF bStartVFD1 THEN
	fbVFD1.Start();	
ELSE
	fbVFD1.Stop();
END_IF

//Pump
fbPump1.AnalogSignal := nFreqInPump1;
bCoilPump1 := fbPump1.Coil;
nFreqOutPump1 := fbPump1.ScaledAnalog;
fbPump1.Scale();

IF bStartPump1 THEN
	fbPump1.Start();	
ELSE
	fbPump1.Stop();
END_IF

END_PROGRAM

// ---- 15_Interface_vs_Herencia/FB_NivelSensor.TcPOU
FUNCTION_BLOCK FB_NivelSensor IMPLEMENTS I_Analog
VAR_INPUT
END_VAR
VAR_OUTPUT
END_VAR
VAR
	_MaxValue 		: INT;
	_ScaledAnalog 	: INT;
	_AnalogSignal 	: INT;
END_VAR

{warning 'Agregar implementación de propiedad'}
PROPERTY AnalogSignal : INT
GET
AnalogSignal := _AnalogSignal;
END_GET
SET
_AnalogSignal := AnalogSignal;
END_SET
END_PROPERTY

PROPERTY MaxValue : INT
GET
MaxValue := _MaxValue;
END_GET
SET
_MaxValue := MaxValue;
END_SET
END_PROPERTY

{warning 'Agregar implementación de método'}
METHOD Scale : BOOL
ScaledAnalog := AnalogSignal * MaxValue / 1000;
END_METHOD

{warning 'Agregar implementación de propiedad'}
PROPERTY ScaledAnalog : INT
GET
ScaledAnalog := _ScaledAnalog;
END_GET
SET
_ScaledAnalog := ScaledAnalog;
END_SET
END_PROPERTY

END_FUNCTION_BLOCK

// ---- 15_Interface_vs_Herencia/FB_UltraSonicSensor.TcPOU
FUNCTION_BLOCK FB_UltraSonicSensor EXTENDS FB_NivelSensor
VAR_INPUT
END_VAR
VAR_OUTPUT
END_VAR
VAR

END_VAR

{warning 'Agregar implementación de método'}
METHOD Scale : BOOL
ScaledAnalog := AnalogSignal * MaxValue / 2000;
END_METHOD

END_FUNCTION_BLOCK

// ---- 15_Interface_vs_Herencia/FB_VFD.TcPOU
FUNCTION_BLOCK FB_VFD IMPLEMENTS I_Analog, I_Run
VAR_INPUT
END_VAR
VAR_OUTPUT
END_VAR
VAR
	_Coil 			: BOOL;
	_AnalogSignal 	: INT;
	_ScaledAnalog 	: INT;
END_VAR

{warning 'Agregar implementación de propiedad'}
PROPERTY AnalogSignal : INT
GET
AnalogSignal := _AnalogSignal;
END_GET
SET
_AnalogSignal := AnalogSignal;
END_SET
END_PROPERTY

{warning 'Agregar implementación de propiedad'}
PROPERTY Coil : BOOL
GET
Coil := _Coil;
END_GET
SET
_Coil := Coil;
END_SET
END_PROPERTY

{warning 'Agregar implementación de método'}
METHOD Scale : BOOL
ScaledAnalog := AnalogSignal * 200;
END_METHOD

{warning 'Agregar implementación de propiedad'}
PROPERTY ScaledAnalog : INT
GET
ScaledAnalog := _ScaledAnalog;
END_GET
SET
_ScaledAnalog := ScaledAnalog;
END_SET
END_PROPERTY

{warning 'Agregar implementación de método'}
METHOD Start : BOOL
Coil := true;
END_METHOD

{warning 'Agregar implementación de método'}
METHOD Stop : BOOL
Coil := false;
END_METHOD

END_FUNCTION_BLOCK

// ---- 15_Interface_vs_Herencia/FB_Pump.TcPOU
FUNCTION_BLOCK FB_Pump EXTENDS FB_VFD
VAR_INPUT
END_VAR
VAR_OUTPUT
END_VAR
VAR
END_VAR

{warning 'Agregar implementación de método'}
METHOD Scale : BOOL
ScaledAnalog := AnalogSignal * 100;
END_METHOD

END_FUNCTION_BLOCK

// ---- 17_Otros_Operadores_1/_17_Otros_Operadores1.TcPOU
PROGRAM _17_Otros_Operadores1
VAR
	pEstructura : POINTER TO ST_Estructura;
	struNew     : BOOL;
END_VAR
VAR
	pSTRING  : POINTER TO STRING;
	bNew     : BOOL;
END_VAR	
VAR CONSTANT
	cLength  : UINT := 150;
END_VAR
VAR
	StruDelete  : BOOL;
END_VAR

// Ejemplos de los Operadores __NEW y  __DELETE
IF struNew AND (pEstructura = 0) THEN
	pEstructura := __NEW(ST_Estructura);	
	struNew := FALSE;
END_IF

IF bNew THEN
    pSTRING := __NEW(BYTE, cLength);
    bNew    := FALSE;
END_IF

IF StruDelete THEN
	 __DELETE(pEstructura);	
	 __DELETE(pSTRING);	
	StruDelete := FALSE;
END_IF

END_PROGRAM

// ---- 18_Otros_Operadores_2/_18_Otros_Operadores2.TcPOU
PROGRAM _18_Otros_Operadores2


QUERYPOINTER();
TRY_CATCH();
VARINFO();
TestAndSet1();

END_PROGRAM

// ---- 18_Otros_Operadores_2/__QUERYPOINTER/QUERYPOINTER.TcPOU
PROGRAM QUERYPOINTER
//__QUERYPOINTER
VAR
    iDerived   : I_Derived;
    fbVariante : FB_Variante;
    bResult    : BOOL;
    bTest      : BOOL;
    pFB        : POINTER TO FB_Variante;
END_VAR

//__QUERYPOINTER
iDerived := fbVariante;
bResult  := __QUERYPOINTER(iDerived, pFB);

IF bResult THEN
    bTest := pFB^.Derived();
END_IF

END_PROGRAM

// ---- 18_Otros_Operadores_2/__QUERYPOINTER/FB_Variante.TcPOU
FUNCTION_BLOCK FB_Variante IMPLEMENTS I_Derived
VAR_INPUT
END_VAR
VAR_OUTPUT
END_VAR
VAR
END_VAR

{warning 'add method implementation '}
METHOD Base : BOOL
END_METHOD

{warning 'add method implementation '}
METHOD Derived : BOOL
END_METHOD

END_FUNCTION_BLOCK

// ---- 18_Otros_Operadores_2/__TRY__CATCH/TRY_CATCH.TcPOU
PROGRAM TRY_CATCH
//__TRY, __CATCH, __FINALLY, __ENDTRY
VAR
    nCounter1          : INT;
    nCounter2          : INT;
    nCounter_TRY1      : INT;
    nCounter_TRY2      : INT;
    nCounter_CATCH     : INT;    
    nCounter_FINALLY   : INT;
 
    exc                : __SYSTEM.ExceptionCode;
    lastExc            : __SYSTEM.ExceptionCode;
 
    pSample            : POINTER TO BOOL;
    bVar               : BOOL;
    nSample            : INT := 100;
    nDivisor           : INT;
END_VAR

//// -- !!! Available FROM TC3.1 build 4024 FOR 32-BIT runtime systems !!!
////__TRY, __CATCH, __FINALLY, __ENDTRY 
//// Counter 1
//nCounter1 := nCounter1 + 1;
 
//// TRY-CATCH block
//__TRY
//    nCounter_TRY1 := nCounter_TRY1 + 1;
//    pSample^      := TRUE;                // 1. cycle: null pointer access leads to "access violation" exception
//    nSample       := nSample/nDivisor;    // 2. cycle: division by zero leads to "divide by zero" exception
//    nCounter_TRY2 := nCounter_TRY2 + 1;
 
//__CATCH(exc)
//    nCounter_CATCH    := nCounter_CATCH + 1;
 
//    // Exception logging
//    lastExc := exc;
//    F_SaveExceptionCode(excInput := exc);
 
//    // Correct the faulty variable values
//    IF (exc = __SYSTEM.ExceptionCode.RTSEXCPT_ACCESS_VIOLATION) AND (pSample = 0) THEN
//        pSample  := ADR(bVar);
// ELSIF ((exc = __SYSTEM.ExceptionCode.RTSEXCPT_DIVIDEBYZERO) OR (exc = __SYSTEM.ExceptionCode.RTSEXCPT_FPU_DIVIDEBYZERO)) AND (nDivisor = 0) THEN
//        nDivisor := 1;
//    END_IF
 
//__FINALLY
//    nCounter_FINALLY := nCounter_FINALLY + 1;
 
//__ENDTRY
 
//// Counter 2
//nCounter2 := nCounter2 + 1;

END_PROGRAM

// ---- 18_Otros_Operadores_2/__VARINFO/VARINFO.TcPOU
PROGRAM VARINFO

VAR
    MyVarInfo : __SYSTEM.VAR_INFO;
    nVar      : INT;
END_VAR

MyVarInfo := __VARINFO(nVar);

END_PROGRAM

// ---- 18_Otros_Operadores_2/TestAndSet/TestAndSet1.TcPOU
PROGRAM TestAndSet1
VAR
    nLocalBlockedCounter : DINT;
END_VAR

IF TestAndSet(GVL.bGlobalTestFlag) THEN
    (* bGlobalTestFlag was FALSE, nobody was blocking, NOW
    bGlobalTestFlag is set to TRUE and blocking others *)
    
    (* ... *)
    
    (* remove blocking by resetting the flag *) 
    GVL.bGlobalTestFlag := FALSE;
ELSE
    (* bGlobalTestFlag was TRUE, somebody is blocking *)
    nLocalBlockedCounter := nLocalBlockedCounter + 1;
    
    (* ... *)
END_IF

END_PROGRAM

// ---- 19_ExST/_19_ExST.TcPOU
PROGRAM _19_ExST
VAR
	myVar: INT;
	myVar1: INT;
	myVar2: INT;
	
	b: BOOL;
	i: INT;	
	btrig : F_TRIG;
	counter: INT;
	
	bVar1: BOOL;
	bVar2: BOOL;
	
	bVar11: BOOL;
	bVar22: BOOL;
	
	bVar: BOOL;
	bVarS: BOOL;
	bVarR: BOOL;
	
	bVara: BOOL;
	bVarb: BOOL;
	bVarc: BOOL;
	
	bMyVar1: BOOL;
	bMyVar2: BOOL;
	bmyTimer : BOOL;
	myTimer : TON;
	

END_VAR

myVar := myVar1 := myVar2 + 26 ; 

IF b := (i = 1) THEN i := i + 1; END_IF	

btrig(CLK:=b);

IF btrig.Q THEN
	counter := counter + 1;
END_IF

bVar1 S= bVar2;

bVar11 R= bVar22;

bVar S= bVarS R= bVarR;

bVara R= bVarb S= bVarc;

myTimer(IN:= bmyTimer , PT:= T#2S );

bMyVar1 S= bMyVar2 R= myTimer.Q;

END_PROGRAM

// ---- 24_SOLID_SRP/_24_SOLID_SRP.TcPOU
PROGRAM _24_SOLID_SRP
VAR
	stRaul 						: ST_Empleado := (Nombre:= 'Raul', Apellido:= 'Gonzalez', CorreoElectronico:= 'micorreo@correo.com');
	Empleado_1 					: FB_Empleado(stRaul);
	
	stHorario_Raul 				: ST_Horario := (HoraEntrada := DT#2023-1-1-8:0:0, HoraSalida := DT#2023-1-1-17:0:0);
	stRegistroDeTiempoEmpleado 	: ST_RegistroDeTiempoEmpleado := (stEmpleado:= stRaul, stHorario:= stHorario_Raul);
	RegistroDeTiempoEmpleado_1 : FB_RegistroDeTiempo(stRegistroDeTiempoEmpleado);
	
	
END_VAR

END_PROGRAM

// ---- 24_SOLID_SRP/Clases_SRP/FB_RegistroDeTiempo.TcPOU
FUNCTION_BLOCK FB_RegistroDeTiempo
VAR_INPUT
	stEmpleado : ST_Empleado; // instancia de la función Empleado
    stHorario  : ST_Horario;
END_VAR
VAR_OUTPUT
END_VAR
VAR
	_RegistroDeTiempo : ST_RegistroDeTiempoEmpleado;
END_VAR

PROPERTY Empleado : ST_Empleado;
GET
END_GET
SET
END_SET
END_PROPERTY

METHOD FB_init : BOOL
VAR_INPUT
	bInitRetains : BOOL; // if TRUE, the retain variables are initialized (warm start / cold start)
	bInCopyCode : BOOL;  // if TRUE, the instance afterwards gets moved into the copy code (online change)
	RegistroDeTiempo : ST_RegistroDeTiempoEmpleado;
END_VAR
_RegistroDeTiempo := RegistroDeTiempo;
END_METHOD

PROPERTY HoraEntrada : DATE_AND_TIME
GET
END_GET
SET
END_SET
END_PROPERTY

PROPERTY HoraSalida : DATE_AND_TIME
GET
END_GET
SET
END_SET
END_PROPERTY

END_FUNCTION_BLOCK

// ---- 25_SOLID_OCP/_25_SOLID_OCP.TcPOU
PROGRAM _25_SOLID_OCP
VAR
	Audi_A8 : FB_Coche;
	Audi_A8_Velocidad :REAL;
	Audi_A8_VelocidadMaxima : REAL;
	
	Suzuki_Ninja : FB_Moto;
	Suzuki_Ninja_Velocidad :REAL;
	Suzuki_Ninja_Aceleracion :REAL;
END_VAR

//Llamada al objeto Audi_A8.
Audi_A8();
//Este metodo es heredado de la clase Vehiculo.
Audi_A8_Velocidad := Audi_A8.getVelocidad(); 
//Este método es propio de la clase Coche.
Audi_A8_VelocidadMaxima := Audi_A8.getVelocidadMaxima();

//Llamada al objeto Suzuki Ninja.
Suzuki_Ninja();
//Este metodo es heredado de la clase Vehiculo
Suzuki_Ninja_Velocidad := Suzuki_Ninja.getVelocidad();
//Este método es propio de la clase Moto.
Suzuki_Ninja_Aceleracion := Suzuki_Ninja.getAceleracion();

END_PROGRAM

// ---- 25_SOLID_OCP/Clases_OCP/FB_Coche.TcPOU
FUNCTION_BLOCK FB_Coche EXTENDS FB_Vehiculo
VAR_INPUT
	velocidadMaxima : REAL;
END_VAR
VAR_OUTPUT
END_VAR
VAR
END_VAR

METHOD getVelocidadMaxima : REAL
VAR_INPUT
END_VAR
getVelocidadMaxima := velocidadMaxima;
END_METHOD

END_FUNCTION_BLOCK

// ---- 25_SOLID_OCP/Clases_OCP/FB_Vehiculo.TcPOU
FUNCTION_BLOCK FB_Vehiculo
VAR_INPUT
	velocidad : REAL;
END_VAR
VAR_OUTPUT
END_VAR
VAR
END_VAR

METHOD getVelocidad : REAL
VAR_INPUT
END_VAR
getVelocidad := velocidad;
END_METHOD

END_FUNCTION_BLOCK

// ---- 25_SOLID_OCP/Clases_OCP/FB_Moto.TcPOU
FUNCTION_BLOCK FB_Moto EXTENDS FB_Vehiculo
VAR_INPUT
	aceleracion : REAL;
END_VAR
VAR_OUTPUT
END_VAR
VAR
END_VAR

METHOD getAceleracion : REAL
VAR_INPUT
END_VAR
getAceleracion := aceleracion;
END_METHOD

END_FUNCTION_BLOCK

// ---- 26_SOLID_LSP/_26_SOLID_LSP.TcPOU
PROGRAM _26_SOLID_LSP
VAR
	Audi_A8 : Coche1;
	Audi_A8_Velocidad_Desada :REAL;
	Audi_A8_Velocidad :REAL;
	
	Suzuki_Ninja: Moto1;
	Suzuki_Ninja_Velocidad_Deseada :REAL;
	Suzuki_Ninja_Velocidad :REAL;
	
	Conductor_Juan : Conductor;
	Conductor_Juan_Velocidad_Deseada :REAL;
	Conductor_Juan_Velocidad : REAL;
	Vehiculo_Seleccionado_Audi_A8 : BOOL;
END_VAR

Audi_A8_Velocidad := Audi_A8.Mover(Audi_A8_Velocidad_Desada);

Suzuki_Ninja_Velocidad := Suzuki_Ninja.Mover(Suzuki_Ninja_Velocidad_Deseada);

IF Vehiculo_Seleccionado_Audi_A8 = TRUE THEN
	Conductor_Juan(vehiculo:= Audi_A8);
ELSE
	Conductor_Juan(vehiculo:= Suzuki_Ninja);
END_IF

Conductor_Juan_Velocidad := Conductor_Juan.Mover(Conductor_Juan_Velocidad_Deseada);

END_PROGRAM

// ---- 26_SOLID_LSP/Clases_LSP/Coche1.TcPOU
FUNCTION_BLOCK Coche1 EXTENDS Vehiculo
VAR_INPUT
	velocidadMaxima : REAL;
END_VAR
VAR_OUTPUT
END_VAR
VAR
END_VAR


METHOD Mover : REAL
VAR_INPUT
	Velocidad_Deseada : REAL;
END_VAR
Mover := Velocidad_Deseada * velocidadMaxima;
END_METHOD

END_FUNCTION_BLOCK

// ---- 26_SOLID_LSP/Clases_LSP/Vehiculo.TcPOU
FUNCTION_BLOCK Vehiculo IMPLEMENTS I_Mover


METHOD Mover : REAL
VAR_INPUT
	Velocidad_Deseada : REAL;
END_VAR
Mover := Velocidad_Deseada;
END_METHOD

END_FUNCTION_BLOCK

// ---- 26_SOLID_LSP/Clases_LSP/Moto1.TcPOU
FUNCTION_BLOCK Moto1 EXTENDS Vehiculo
VAR_INPUT
	Aceleracion : REAL;
END_VAR
VAR_OUTPUT
END_VAR
VAR
END_VAR


METHOD Mover : REAL
VAR_INPUT
	Velocidad_Deseada : REAL;
END_VAR
Mover := Velocidad_Deseada * Aceleracion ;
END_METHOD

END_FUNCTION_BLOCK

// ---- 26_SOLID_LSP/Clases_LSP/Conductor.TcPOU
FUNCTION_BLOCK Conductor
VAR_INPUT
	vehiculo : REFERENCE TO Vehiculo(THIS^); // referencia a la clase base Vehiculo
END_VAR
VAR_OUTPUT
END_VAR
VAR
END_VAR

METHOD Mover : REAL
VAR_INPUT
	Velocidad_Deseada : REAL;
END_VAR
Mover := THIS^.vehiculo.Mover(Velocidad_Deseada);
END_METHOD

END_FUNCTION_BLOCK

// ---- 27_SOLID_ISP/_27_SOLID_ISP.TcPOU
PROGRAM _27_SOLID_ISP
VAR
	Patito_feo : Pato;
	Aguila_imperial : Aguila;
	Avestruz_de_cuello_azul : Avestruz;
END_VAR

Patito_feo.Nadar();
Patito_feo.Volar();

Aguila_imperial.Volar();

Avestruz_de_cuello_azul.Correr();

END_PROGRAM

// ---- 27_SOLID_ISP/Clases_ISP/Pato.TcPOU
FUNCTION_BLOCK Pato IMPLEMENTS I_AveVoladora, I_AveNadadora
VAR_INPUT
    velocidad : REAL;
    alturaMaxima : REAL;
    tiempoBuceo : TIME;
END_VAR
VAR
END_VAR


METHOD Nadar : BOOL
Nadar := TRUE;
END_METHOD


METHOD Volar : BOOL
Volar := true;
END_METHOD

END_FUNCTION_BLOCK

// ---- 27_SOLID_ISP/Clases_ISP/Aguila.TcPOU
FUNCTION_BLOCK Aguila IMPLEMENTS I_AveVoladora
VAR_INPUT
    velocidad : REAL;
    alturaMaxima : REAL;
END_VAR
VAR
END_VAR


METHOD Volar : BOOL
Volar:= TRUE;
END_METHOD

END_FUNCTION_BLOCK

// ---- 27_SOLID_ISP/Clases_ISP/Avestruz.TcPOU
FUNCTION_BLOCK Avestruz IMPLEMENTS I_AveCorredora
VAR_INPUT
    velocidad : REAL;
    tiempoCorriendo : TIME;
END_VAR
VAR
END_VAR


METHOD Correr : BOOL
Correr := TRUE;
END_METHOD

END_FUNCTION_BLOCK

// ---- 28_SOLID_DIP/_28_SOLID_DIP.TcPOU
PROGRAM _28_SOLID_DIP
VAR
	Conexion_por_Serial : BOOL;
	Serial: ConexionSerial;
	Conexion_Serial : Dispositivo(conexion:= Serial);
	
	Conexion_por_Ethernet : BOOL;
	Ethernet : ConexionEthernet;
	Conexion_Ethernet : Dispositivo(conexion:= Ethernet);
END_VAR


IF Conexion_por_Serial THEN 
 Conexion_Serial.establecerConexion();
 Conexion_por_Serial:= FALSE;
END_IF

IF Conexion_por_Ethernet THEN 
 Conexion_Ethernet.establecerConexion();
 Conexion_por_Ethernet:= FALSE;
END_IF

END_PROGRAM

// ---- 28_SOLID_DIP/Clases_DIP/ConexionSerial.TcPOU
FUNCTION_BLOCK ConexionSerial IMPLEMENTS I_Conexion

VAR
    udiAdsLogRes: DINT;
END_VAR


METHOD EstablecerConexion : BOOL

UdiAdsLogRes := ADSLOGDINT( msgCtrlMask := ADSLOG_MSGTYPE_HINT OR ADSLOG_MSGTYPE_MSGBOX, 
                            msgFmtStr := 'PLC Mensaje: estamos realizando una conexión por Serial: %d', dintArg:= 1);
END_METHOD

END_FUNCTION_BLOCK

// ---- 28_SOLID_DIP/Clases_DIP/Dispositivo.TcPOU
FUNCTION_BLOCK Dispositivo
VAR
	_conexion : I_Conexion;
END_VAR

METHOD establecerConexion 
VAR_INPUT
END_VAR
_conexion.EstablecerConexion();
END_METHOD

METHOD FB_init : BOOL
VAR_INPUT
	bInitRetains : BOOL; // if TRUE, the retain variables are initialized (warm start / cold start)
	bInCopyCode : BOOL;  // if TRUE, the instance afterwards gets moved into the copy code (online change)
	conexion : I_Conexion;
END_VAR
THIS^._conexion := conexion;
END_METHOD

END_FUNCTION_BLOCK

// ---- 28_SOLID_DIP/Clases_DIP/ConexionEthernet.TcPOU
FUNCTION_BLOCK ConexionEthernet IMPLEMENTS I_Conexion

VAR
    udiAdsLogRes: DINT;
END_VAR


METHOD EstablecerConexion : BOOL

UdiAdsLogRes := ADSLOGDINT( msgCtrlMask := ADSLOG_MSGTYPE_HINT OR ADSLOG_MSGTYPE_MSGBOX, 
                            msgFmtStr := 'PLC Mensaje: estamos realizando una conexión por Ethernet: %d', dintArg:= 1);
END_METHOD

END_FUNCTION_BLOCK

// ---- 32_UML_StateChart/32_POUs/_32_MAIN.TcPOU
(*
### This sample project contains the following elements.

- FB_UML_SC:		This FB represents a simulation to save a text as XML or text format, and to publish it afterwards to a client and to a master.
					The underlying state machine is implemented with the help of UML State Chart.
					
					The behavior is not really programmed.
					Only the wrapper/basic structure of the state machine is implemented. 
						
					Each time, when an ENTRY/DO/EXIT action is called, a correspondent counter variable is increased.

- Visualization:	The visu shows the state of the counters, so that you can see how often an ENTRY/DO/EXIT action has been called. 
					You can use the buttons to switch between the states.
*)
PROGRAM _32_MAIN
VAR
	fbUmlSC	: FB_UML_SC;
END_VAR

fbUmlSC();

END_PROGRAM

// ---- 32_UML_StateChart/32_POUs/FB_UML_SC.TcPOU
FUNCTION_BLOCK FB_UML_SC
VAR
	// Transition condition
	bInitFinished				: BOOL;
	bUseXmlFormat				: BOOL;
	bAllInfoCopiedToFile		: BOOL;
	bSendToMasterFinished		: BOOL;
	bSendToClientFinished		: BOOL;
	
	// Counters
	nCounterInit				: INT;
	nCounterSaveInitSettings	: INT;
	nCounterClearXml			: INT;
	nCounterFillXml				: INT;
	nCounterSaveXml				: INT;
	nCounterClearText			: INT;
	nCounterFillText			: INT;
	nCounterSaveText			: INT;
	nCounterGetMasterID			: INT;
	nCounterGetClientID			: INT;
	nCounterSendToMaster		: INT;
	nCounterSendToClient		: INT;
	
	// Debugging
	bMasterFirst				: BOOL;
	bClientFirst				: BOOL;
END_VAR

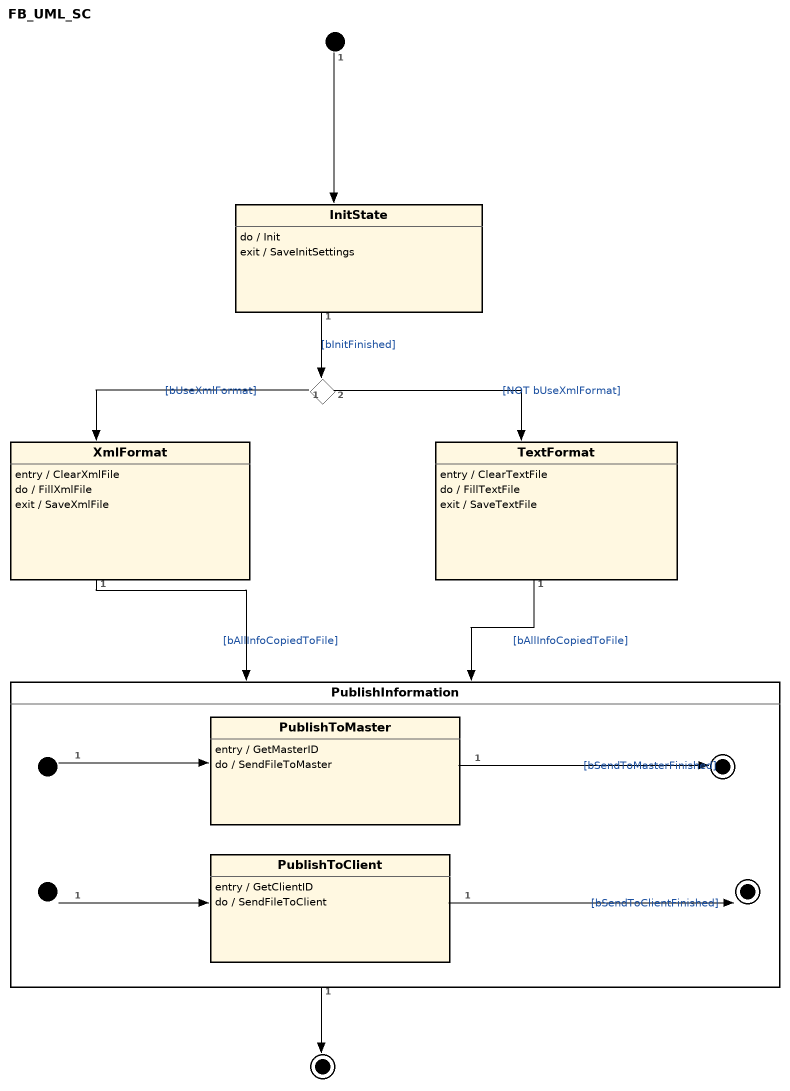
STATECHART FB_UML_SC  // abortable
    START StartState1
    STATE InitState
        do / Init
        exit / SaveInitSettings
    CHOICE ChoiceElement1
    STATE XmlFormat
        entry / ClearXmlFile
        do / FillXmlFile
        exit / SaveXmlFile
    STATE TextFormat
        entry / ClearTextFile
        do / FillTextFile
        exit / SaveTextFile
    COMPOSITE STATE PublishInformation
        REGION Region0 // priority 1
        START StartState2
        STATE PublishToMaster
            entry / GetMasterID
            do / SendFileToMaster
        END EndState2
        StartState2 -> PublishToMaster  // priority 1, on completion
        PublishToMaster -> EndState2 [bSendToMasterFinished] // priority 1
        REGION Region1 // priority 2
        START StartState3
        STATE PublishToClient
            entry / GetClientID
            do / SendFileToClient
        END EndState3
        StartState3 -> PublishToClient  // priority 1, on completion
        PublishToClient -> EndState3 [bSendToClientFinished] // priority 1
    END_STATE
    END EndState1
    StartState1 -> InitState  // priority 1, on completion
    InitState -> ChoiceElement1 [bInitFinished] // priority 1
    ChoiceElement1 -> XmlFormat [bUseXmlFormat] // priority 1
    ChoiceElement1 -> TextFormat [NOT bUseXmlFormat] // priority 2
    XmlFormat -> PublishInformation [bAllInfoCopiedToFile] // priority 1
    TextFormat -> PublishInformation [bAllInfoCopiedToFile] // priority 1
    PublishInformation -> EndState1  // priority 1, on completion
END_STATECHART

METHOD PROTECTED ClearTextFile
VAR_INPUT
END_VAR
nCounterClearText := nCounterClearText + 1;
END_METHOD

METHOD PROTECTED ClearXmlFile
VAR_INPUT
END_VAR
nCounterClearXml := nCounterClearXml + 1;
END_METHOD

METHOD PROTECTED FillTextFile
VAR_INPUT
END_VAR
nCounterFillText := nCounterFillText + 1;
END_METHOD

METHOD PROTECTED FillXmlFile
VAR_INPUT
END_VAR
nCounterFillXml := nCounterFillXml + 1;
END_METHOD

METHOD PROTECTED GetClientID
VAR_INPUT
END_VAR
nCounterGetClientID := nCounterGetClientID + 1;

IF NOT bMasterFirst THEN
	bClientFirst := TRUE;
END_IF
END_METHOD

METHOD PROTECTED GetMasterID
VAR_INPUT
END_VAR
nCounterGetMasterID := nCounterGetMasterID + 1;

IF NOT bClientFirst THEN
	bMasterFirst := TRUE;
END_IF
END_METHOD

METHOD PROTECTED Init
VAR_INPUT
END_VAR
nCounterInit := nCounterInit + 1;
END_METHOD

METHOD PROTECTED SaveInitSettings
VAR_INPUT
END_VAR
nCounterSaveInitSettings := nCounterSaveInitSettings + 1;

bInitFinished 			:= FALSE;
bAllInfoCopiedToFile 	:= FALSE;
bSendToClientFinished 	:= FALSE;
bSendToMasterFinished	:= FALSE;
bMasterFirst			:= FALSE;
bClientFirst			:= FALSE;
END_METHOD

METHOD PROTECTED SaveTextFile
VAR_INPUT
END_VAR
nCounterSaveText := nCounterSaveText + 1;
END_METHOD

METHOD PROTECTED SaveXmlFile
VAR_INPUT
END_VAR
nCounterSaveXml := nCounterSaveXml + 1;
END_METHOD

METHOD PROTECTED SendFileToClient
VAR_INPUT
END_VAR
nCounterSendToClient := nCounterSendToClient + 1;
END_METHOD

METHOD PROTECTED SendFileToMaster
VAR_INPUT
END_VAR
nCounterSendToMaster := nCounterSendToMaster + 1;
END_METHOD

END_FUNCTION_BLOCK

// ---- 07_Herencia_FB/FB_Padre.TcPOU
FUNCTION_BLOCK FB_Padre
VAR_INPUT
	iIn1: INT;
END_VAR
VAR_OUTPUT
	iOut:INT;
END_VAR
VAR
	iPadreVar:INT:= 42;
	iPadreTime: TON:=(in:=TRUE, pt:=T#1S);
END_VAR

iPadreTime();
IF iPadreTime.Q THEN
	iPadreVar:= iPadreVar+iIn1;
	iPadreTime.IN:= FALSE;
ELSE
	iPadreTime.IN:= TRUE;
END_IF

METHOD mDouble : INT
VAR_INPUT
END_VAR
mDouble:= iIn1+iIn1;
END_METHOD

METHOD mMultiply : INT
VAR_INPUT
END_VAR
mMultiply := iIn1*5;
END_METHOD

END_FUNCTION_BLOCK

// ---- 12_Concepto Keyword Abstract/ConcreteLoadCell.TcPOU
FUNCTION_BLOCK PUBLIC ConcreteLoadCell EXTENDS AbstractLoadCell
VAR_INPUT
END_VAR
VAR_OUTPUT
END_VAR
VAR
END_VAR

END_FUNCTION_BLOCK

// ---- 16_17_Interface_vs_Herencia/FB_MyLight1.TcPOU
FUNCTION_BLOCK FB_MyLight1 EXTENDS FB_Light IMPLEMENTS I_Delayable, I_Dimmable
VAR_INPUT
	bRecallMinLevel			:	BOOL;
	bSetControlLevel		:	BOOL;
	nSetControlLevel		:	BYTE;
END_VAR
VAR_OUTPUT
	nControl				:	BYTE;
END_VAR
VAR
	rtrigRecallMinLevel		:	R_TRIG;
	rtrigSetControlLevel	:	R_TRIG;
	fbDimmingLight			:	FB_DimmingLight;
	fbDelayedLight			:	FB_DelayedLight;
	_nControlLevel			:	BYTE;
END_VAR

rtrigOn(CLK := bOn);
IF (rtrigOn.Q) THEN
	M_On();
END_IF

rtrigOff(CLK := bOff);
IF (rtrigOff.Q) THEN
	M_Off();
END_IF

rtrigRecallMinLevel(CLK := bRecallMinLevel);
IF (rtrigRecallMinLevel.Q) THEN
	M_RecallMinLevel();
END_IF

rtrigSetControlLevel(CLK := bSetControlLevel);
IF (rtrigSetControlLevel.Q) THEN
	M_SetControlLevel(nSetControlLevel);
END_IF

fbDimmingLight();
fbDelayedLight();
_bControlLevel := fbDelayedLight.bControlLevel;
IF (_bControlLevel) THEN
	_nControlLevel := fbDimmingLight.nControlLevel;
ELSE
	_nControlLevel := 0;		
END_IF

bControl := bControlLevel;
nControl := nControlLevel;

PROPERTY bControlLevel : BOOL
GET
bControlLevel := _bControlLevel;
END_GET
SET
END_SET
END_PROPERTY

METHOD M_Off
fbDimmingLight.M_Off();
fbDelayedLight.M_Off();
END_METHOD

METHOD M_On
fbDimmingLight.M_On();
fbDelayedLight.M_On();
END_METHOD

METHOD M_RecallMinLevel
fbDimmingLight.M_RecallMinLevel();
fbDelayedLight.M_On();
END_METHOD

METHOD M_SetControlLevel
VAR_INPUT
	nControlLevel: BYTE;
END_VAR
fbDimmingLight.M_SetControlLevel(nControlLevel);
IF (nControlLevel = 0) THEN
	fbDelayedLight.M_Off();
ELSE
	fbDelayedLight.M_On();
END_IF
END_METHOD

PROPERTY nControlLevel : BYTE
GET
nControlLevel := _nControlLevel;
END_GET
SET
END_SET
END_PROPERTY

PROPERTY nMaxLevel : BYTE
GET
nMaxLevel := THIS^.fbDimmingLight.nMaxLevel;
END_GET
SET
THIS^.fbDimmingLight.nMaxLevel := nMaxLevel;
END_SET
END_PROPERTY

PROPERTY nMinLevel : BYTE
GET
nMinLevel := THIS^.fbDimmingLight.nMinLevel;
END_GET
SET
THIS^.fbDimmingLight.nMaxLevel := nMaxLevel;
END_SET
END_PROPERTY

PROPERTY tOffDelay : TIME
GET
END_GET
SET
END_SET
END_PROPERTY

PROPERTY tOnDelay : TIME
GET
END_GET
SET
END_SET
END_PROPERTY

END_FUNCTION_BLOCK

// ---- 16_17_Interface_vs_Herencia/PLC-Library/Clases/FB_Light.TcPOU
FUNCTION_BLOCK PUBLIC FB_Light IMPLEMENTS I_Light
VAR_INPUT
	bOn					:	BOOL;
	bOff				:	BOOL;
END_VAR
VAR_OUTPUT
	bControl			:	BOOL;
END_VAR
VAR
	rtrigOn				:	R_TRIG;
	rtrigOff			:	R_TRIG;
	_bControlLevel		:	BOOL;
END_VAR

rtrigOn(CLK := bOn);
IF (rtrigOn.Q) THEN
	M_On();
END_IF

rtrigOff(CLK := bOff);
IF (rtrigOff.Q) THEN
	M_Off();
END_IF

bControl := bControlLevel;

PROPERTY bControlLevel : BOOL
GET
bControlLevel := _bControlLevel;
END_GET
SET
END_SET
END_PROPERTY

METHOD PUBLIC M_Off
_bControlLevel := FALSE;
END_METHOD

METHOD PUBLIC M_On
_bControlLevel := TRUE;
END_METHOD

END_FUNCTION_BLOCK

// ---- 16_17_Interface_vs_Herencia/PLC-Library/FB_MyLight.TcPOU
FUNCTION_BLOCK FB_MyLight EXTENDS FB_Light IMPLEMENTS I_Delayable, I_Dimmable
VAR_INPUT
	bRecallMinLevel			:	BOOL;
	bSetControlLevel		:	BOOL;
	nSetControlLevel		:	BYTE;
END_VAR
VAR_OUTPUT
	nControl				:	BYTE;
END_VAR
VAR
	rtrigRecallMinLevel		:	R_TRIG;
	rtrigSetControlLevel	:	R_TRIG;
	fbDimmingLight			:	FB_DimmingLight;
	fbDelayedLight			:	FB_DelayedLight;
	_nControlLevel			:	BYTE;
END_VAR

rtrigOn(CLK := bOn);
IF (rtrigOn.Q) THEN
	M_On();
END_IF

rtrigOff(CLK := bOff);
IF (rtrigOff.Q) THEN
	M_Off();
END_IF

rtrigRecallMinLevel(CLK := bRecallMinLevel);
IF (rtrigRecallMinLevel.Q) THEN
	M_RecallMinLevel();
END_IF

rtrigSetControlLevel(CLK := bSetControlLevel);
IF (rtrigSetControlLevel.Q) THEN
	M_SetControlLevel(nSetControlLevel);
END_IF

fbDimmingLight();
fbDelayedLight();
_bControlLevel := fbDelayedLight.bControlLevel;
IF (_bControlLevel) THEN
	_nControlLevel := fbDimmingLight.nControlLevel;
ELSE
	_nControlLevel := 0;		
END_IF

bControl := bControlLevel;
nControl := nControlLevel;

PROPERTY bControlLevel : BOOL
GET
bControlLevel := _bControlLevel;
END_GET
SET
END_SET
END_PROPERTY

METHOD M_Off
fbDimmingLight.M_Off();
fbDelayedLight.M_Off();
END_METHOD

METHOD M_On
fbDimmingLight.M_On();
fbDelayedLight.M_On();
END_METHOD

METHOD M_RecallMinLevel
fbDimmingLight.M_RecallMinLevel();
fbDelayedLight.M_On();
END_METHOD

METHOD M_SetControlLevel
VAR_INPUT
	nControlLevel: BYTE;
END_VAR
fbDimmingLight.M_SetControlLevel(nControlLevel);
IF (nControlLevel = 0) THEN
	fbDelayedLight.M_Off();
ELSE
	fbDelayedLight.M_On();
END_IF
END_METHOD

PROPERTY nControlLevel : BYTE
GET
nControlLevel := _nControlLevel;
END_GET
SET
END_SET
END_PROPERTY

PROPERTY nMaxLevel : BYTE
GET
nMaxLevel := THIS^.fbDimmingLight.nMaxLevel;
END_GET
SET
THIS^.fbDimmingLight.nMaxLevel := nMaxLevel;
END_SET
END_PROPERTY

PROPERTY nMinLevel : BYTE
GET
nMinLevel := THIS^.fbDimmingLight.nMinLevel;
END_GET
SET
THIS^.fbDimmingLight.nMaxLevel := nMaxLevel;
END_SET
END_PROPERTY

PROPERTY tOffDelay : TIME
GET
END_GET
SET
END_SET
END_PROPERTY

PROPERTY tOnDelay : TIME
GET
END_GET
SET
END_SET
END_PROPERTY

END_FUNCTION_BLOCK

// ---- 16_17_Interface_vs_Herencia/Tests/P_DimmingLight_Test_CFC.TcPOU
PROGRAM P_DimmingLight_Test_CFC
VAR
	fbDimmingLight		:	FB_DimmingLight;
	bOn					:	BOOL;
	bOff				:	BOOL;
	bRecallMinLevel		:	BOOL;
	bSetControlLevel	:	BOOL;
	nSetControlLevel	:	BYTE;
	bControlLevel		:	BOOL;
	nControlLevel		:	BYTE;
END_VAR

fbDimmingLight(
    bOn := bOn,
    bOff := bOff,
    bRecallMinLevel := bRecallMinLevel,
    bSetControlLevel := bSetControlLevel,
    nSetControlLevel := nSetControlLevel); // FB_DimmingLight
bControlLevel := fbDimmingLight.bControl;
nControlLevel := fbDimmingLight.nControl;

END_PROGRAM

// ---- 16_17_Interface_vs_Herencia/Tests/P_Light_Test_CFC.TcPOU
PROGRAM P_Light_Test_CFC
VAR
	fbLight				:	FB_Light;
	bOn					:	BOOL;
	bOff				:	BOOL;
	bControlLevel		:	BOOL;
END_VAR

fbLight(bOn := bOn, bOff := bOff); // FB_Light
bControlLevel := fbLight.bControl;

END_PROGRAM

// ---- 16_17_Interface_vs_Herencia/Tests/P_Light_Test_ST.TcPOU
PROGRAM P_Light_Test_ST
VAR
	fbLight				:	FB_Light;
	bOn					:	BOOL;
	bOff				:	BOOL;
	bControlLevel		:	BOOL;	
END_VAR

fbLight();

IF (bOn) THEN
	fbLight.M_On();
	bOn := FALSE;
END_IF
IF (bOff) THEN
	fbLight.M_Off();
	bOff := FALSE;
END_IF

bControlLevel := fbLight.bControlLevel;

END_PROGRAM

// ---- 16_17_Interface_vs_Herencia/Tests/P_MyLight_Test_CFC.TcPOU
PROGRAM P_MyLight_Test_CFC
VAR
	fbMyLight			:	FB_MyLight1;
	bOn					:	BOOL;
	bOff				:	BOOL;
	bRecallMinLevel		:	BOOL;
	bSetControlLevel	:	BOOL;
	nSetControlLevel	:	BYTE;
	bControlLevel		:	BOOL;
	nControlLevel		:	BYTE;
END_VAR

bControlLevel := fbMyLight.bControl;
nControlLevel := fbMyLight.nControl;
fbMyLight(
    bOn := bOn,
    bOff := bOff,
    bRecallMinLevel := bRecallMinLevel,
    bSetControlLevel := bSetControlLevel,
    nSetControlLevel := nSetControlLevel); // FB_MyLight1

END_PROGRAM

// ---- 16_17_Interface_vs_Herencia/Tests/P_MyLight_Test_ST.TcPOU
PROGRAM P_MyLight_Test_ST
VAR
	fbMyLight			:	FB_MyLight1;
	bOn					:	BOOL;
	bOff				:	BOOL;
	bRecallMinLevel		:	BOOL;
	bSetControlLevel	:	BOOL;
	nSetControlLevel	:	BYTE;
	bControlLevel		:	BOOL;
	nControlLevel		:	BYTE;
END_VAR

fbMyLight();

IF (bOn) THEN
	fbMyLight.M_On();
	bOn := FALSE;
END_IF
IF (bOff) THEN
	fbMyLight.M_Off();
	bOff := FALSE;
END_IF
IF (bRecallMinLevel) THEN
	fbMyLight.M_RecallMinLevel();
	bRecallMinLevel := FALSE;
END_IF
IF (bSetControlLevel) THEN
	fbMyLight.M_SetControlLevel(nSetControlLevel);
	bSetControlLevel := FALSE;
END_IF

bControlLevel := fbMyLight.bControlLevel;
nControlLevel := fbMyLight.nControlLevel;

END_PROGRAM

// ---- 16_17_Interface_vs_Herencia/Tests/P_RoomController_Test_CFC.TcPOU
PROGRAM P_RoomController_Test_CFC
VAR
	fbRoomController	:	FB_RoomController;
	fbmyLight			:	FB_MyLight1;
	fbDelayedLight		:	FB_DelayedLight;
	fbDimmingLight		:	FB_DimmingLight;
	bAllOn				:	BOOL;
	bAllOff				:	BOOL;
	bAllCallMinLevel	:	BOOL;
	aControlLevel		:	ARRAY [1..3] OF BOOL;
	aDimmLevel			:	ARRAY [1..3] OF BYTE;
END_VAR

fbRoomController(
    bAllOn := bAllOn,
    bAllOff := bAllOff,
    bAllCallMinLevel := bAllCallMinLevel,
    refLight01 := fbMyLight,
    refLight02 := fbDelayedLight,
    refLight03 := fbDimmingLight); // FB_RoomController
aControlLevel := fbRoomController.aControlLevel;
aDimmLevel := fbRoomController.aDimmLevel;

END_PROGRAM

// ---- 16_17_Interface_vs_Herencia/Tests/P_RoomController_Test_ST.TcPOU
PROGRAM P_RoomController_Test_ST
VAR
	fbRoomController	:	FB_RoomController;
	fbMyLight			:	FB_MyLight1;
	fbDelayedLight		:	FB_DelayedLight;
	fbDimmingLight		:	FB_DimmingLight;
	bAllOn				:	BOOL;
	bAllOff				:	BOOL;
	bAllCallMinLevel	:	BOOL;
	aControlLevel		:	ARRAY [1..3] OF BOOL;
	aDimmLevel			:	ARRAY [1..3] OF BYTE;
END_VAR

fbRoomController(bAllOn	:= bAllOn,
				 bAllOff := bAllOff,
				 bAllCallMinLevel := bAllCallMinLevel,
				 refLight01 := fbMyLight,
				 refLight02 := fbDelayedLight,
				 refLight03 := fbDimmingLight,
				 aControlLevel => aControlLevel,
				 aDimmLevel => aDimmLevel);

END_PROGRAM

// ---- 18_Otros_Operadores_2/__TRY__CATCH/F_SaveExceptionCode.TcPOU
FUNCTION F_SaveExceptionCode : BOOL
VAR_INPUT
    excInput           : __SYSTEM.ExceptionCode;
END_VAR

// Log the thrown exception into the global exception history array
IF GVL_Exc.nExcIndex <= GVL_Exc.cMaxExc THEN
    GVL_Exc.aExceptionHistory[GVL_Exc.nExcIndex] := excInput;
    GVL_Exc.nExcIndex := GVL_Exc.nExcIndex + 1;
END_IF

END_FUNCTION

// ---- 30_UML_ClassDiagram/Persona.TcPOU
FUNCTION_BLOCK Persona
VAR_INPUT
END_VAR
VAR_OUTPUT
END_VAR
VAR
END_VAR

METHOD Comer
VAR_INPUT
END_VAR
END_METHOD

PROPERTY DNI : string
GET
END_GET
SET
END_SET
END_PROPERTY

END_FUNCTION_BLOCK

// ---- 30_UML_ClassDiagram/Profesor.TcPOU
FUNCTION_BLOCK Profesor EXTENDS Persona IMPLEMENTS ITF_Profesor
VAR_INPUT
END_VAR
VAR_OUTPUT
END_VAR
VAR
	_Nombre: STRING;
END_VAR

METHOD DarClases
VAR_INPUT
END_VAR
END_METHOD

{warning 'Agregar implementación de método'}
METHOD Fichar
END_METHOD

PROPERTY Nombre : String
GET
END_GET
SET
END_SET
END_PROPERTY

{warning 'Agregar implementación de propiedad'}
PROPERTY Salida : INT
GET
END_GET
SET
END_SET
END_PROPERTY

END_FUNCTION_BLOCK

// ---- 31_UML_relaciones/Corazon.TcPOU
FUNCTION_BLOCK Corazon
VAR_INPUT
END_VAR
VAR_OUTPUT
END_VAR
VAR
	VarHumano: Humano;
	pHumano: POINTER TO Humano;
	pHumano16: REFERENCE TO Humano;
END_VAR

END_FUNCTION_BLOCK

// ---- 31_UML_relaciones/Humano.TcPOU
FUNCTION_BLOCK Humano IMPLEMENTS I_Humano
VAR_INPUT
END_VAR
VAR_OUTPUT
END_VAR
VAR
END_VAR

{warning 'Agregar implementación de método'}
METHOD Correr
END_METHOD

{warning 'Agregar implementación de propiedad'}
PROPERTY Nombre : STRING
GET
END_GET
SET
END_SET
END_PROPERTY

END_FUNCTION_BLOCK

// ---- 31_UML_relaciones/Hombre.TcPOU
FUNCTION_BLOCK Hombre EXTENDS Humano
VAR_INPUT
END_VAR
VAR_OUTPUT
END_VAR
VAR
END_VAR

END_FUNCTION_BLOCK

// ---- 31_UML_relaciones/Sangre.TcPOU
FUNCTION_BLOCK Sangre
VAR_INPUT
END_VAR
VAR_OUTPUT
END_VAR
VAR
	VarHumano: Humano;
END_VAR

END_FUNCTION_BLOCK

// ---- 32_UML_StateChart/Kaffemaschine.TcPOU
{attribute 'no-analysis' := ''}
{attribute 'reduced_bp_set' := ''}
PROGRAM Kaffemaschine
VAR
	bMakeCoffee: BOOL := FALSE;
	bShutDown: BOOL := FALSE;
	bPowerUp: BOOL := FALSE;
	nGrind: INT := 0;
	nHeat: INT := 20;
	nFoam: INT := 0;
	{attribute 'implicit_state_chart_struct' := ''}
	UML_SC_Kaffemaschine: _UML_SC_7cc42eb0dc6d4e02ab5b1296bec80ed6;
	{attribute 'implicit_state_chart_struct' := ''}
	UML_SC_ActHeat: _UML_SC_9e3c3d30f6c84991be9f932f948dff00;
END_VAR

ACTION ActDo:
nGrind := nGrind + 10;
END_ACTION

ACTION ActEntry:

END_ACTION

ACTION ActFoam:
nFoam := nFoam + 5;
END_ACTION

ACTION ActHeat:

END_ACTION

ACTION ActShutdown:
bShutDown := FALSE;
bPowerUp := FALSE;
END_ACTION

ACTION CoffeeReady:
bMakeCoffee := FALSE;
nGrind := 0;
nHeat := 20;
nFoam := 0;
END_ACTION

END_PROGRAM

